DATA_BLOCK "HMI animation"	// DB 60
TITLE = HMI ANIMATION DATA BLOCK
AUTHOR : Milesi
VERSION : 0.1
  STRUCT
   Take_up_unit : STRUCT
    DB60_DBX0_0 : BOOL ;	//General alarm
    DB60_DBX0_1 : BOOL ;	//Driven pintle emergency
    DB60_DBX0_2 : BOOL ;	//Idle pintle emergency
    DB60_DBX0_3 : BOOL ;	//Bobbin down
    DB60_DBX0_4 : BOOL ;	//Speed reference right inversion
    DB60_DBX0_5 : BOOL ;	//Speed reference left inversion
    DB60_DBX0_6 : BOOL ;
    DB60_DBX0_7 : BOOL ;
    DB60_DBB1 : BYTE ;	//Motor status
    DB60_DBB2 : BYTE ;	//Motor blower status
    DB60_DBB3 : BYTE ;	//Traverse motor status
    DB60_DBB4 : BYTE ;	//Traverse motor blower status
    DB60_DBB5 : BYTE ;	//Bobbin driven pintle motor status
    DB60_DBB6 : BYTE ;	//Bobbin idle pintle motor status
    DB60_DBB7 : BYTE ;	//Bobbin pintle opening-closing motor status
    DB60_DBB8 : BYTE ;
    DB60_DBB9 : BYTE ;
    DB60_DBB10 : BYTE ;
   END_STRUCT ;
   Capstan : STRUCT
    DB60_DBX12_0 : BOOL ;	//General alarm
    DB60_DBX12_1 : BOOL ;	//Cable block open
    DB60_DBX12_2 : BOOL ;
    DB60_DBX12_3 : BOOL ;
    DB60_DBX12_4 : BOOL ;
    DB60_DBX12_5 : BOOL ;
    DB60_DBX12_6 : BOOL ;
    DB60_DBX12_7 : BOOL ;
    DB60_DBB13 : BYTE ;	//Motor status
    DB60_DBB14 : BYTE ;	//Motor blower status
    DB60_DBW16 : INT ;
    DB60_DBW18 : INT ;
    DB60_DBD20 : REAL ;
   END_STRUCT ;
   Lateral_taping_head : STRUCT
    DB60_DBX24_0 : BOOL ;	//General alarm
    DB60_DBX24_1 : BOOL ;
    DB60_DBX24_2 : BOOL ;
    DB60_DBX24_3 : BOOL ;
    DB60_DBX24_4 : BOOL ;
    DB60_DBX24_5 : BOOL ;
    DB60_DBX24_6 : BOOL ;
    DB60_DBX24_7 : BOOL ;
    DB60_DBB25 : BYTE ;	//Motor status
    DB60_DBB26 : BYTE ;	//Motor blower status
    DB60_DBW28 : INT ;
    DB60_DBW30 : INT ;
    DB60_DBD32 : REAL ;
   END_STRUCT ;
   Cage_24 : STRUCT
    DB60_DBX36_0 : BOOL ;	//General alarm
    DB60_DBX36_1 : BOOL ;
    DB60_DBX36_2 : BOOL ;
    DB60_DBX36_3 : BOOL ;
    DB60_DBX36_4 : BOOL ;
    DB60_DBX36_5 : BOOL ;
    DB60_DBX36_6 : BOOL ;
    DB60_DBX36_7 : BOOL ;
    DB60_DBB37 : BYTE ;	//Motor status
    DB60_DBB38 : BYTE ;	//Motor blower status
    DB60_DBB39 : BYTE ;	//Loading motor status
    DB60_DBB40 : BYTE ;
    DB60_DBW42 : INT ;
    DB60_DBD46 : REAL ;
   END_STRUCT ;
   Cage_24_preforming : STRUCT
    DB60_DBX48_0 : BOOL ;	//General alarm
    DB60_DBX48_1 : BOOL ;
    DB60_DBX48_2 : BOOL ;
    DB60_DBX48_3 : BOOL ;
    DB60_DBX48_4 : BOOL ;
    DB60_DBX48_5 : BOOL ;
    DB60_DBX48_6 : BOOL ;
    DB60_DBX48_7 : BOOL ;
    DB60_DBB49 : BYTE ;	//Motor status
    DB60_DBB50 : BYTE ;	//Motor blower status
    DB60_DBW52 : INT ;
    DB60_DBW54 : INT ;
    DB60_DBD56 : REAL ;
   END_STRUCT ;
   Cage_18 : STRUCT
    DB60_DBX60_0 : BOOL ;	//General alarm
    DB60_DBX60_1 : BOOL ;
    DB60_DBX60_2 : BOOL ;
    DB60_DBX60_3 : BOOL ;
    DB60_DBX60_4 : BOOL ;
    DB60_DBX60_5 : BOOL ;
    DB60_DBX60_6 : BOOL ;
    DB60_DBX60_7 : BOOL ;
    DB60_DBB61 : BYTE ;	//Motor status
    DB60_DBB62 : BYTE ;	//Motor blower status
    DB60_DBB63 : BYTE ;	//Loading motor status
    DB60_DBB64 : BYTE ;
    DB60_DBW66 : INT ;
    DB60_DBD68 : REAL ;
   END_STRUCT ;
   Cage_18_preforming : STRUCT
    DB60_DBX72_0 : BOOL ;	//General alarm
    DB60_DBX72_1 : BOOL ;
    DB60_DBX72_2 : BOOL ;
    DB60_DBX72_3 : BOOL ;
    DB60_DBX72_4 : BOOL ;
    DB60_DBX72_5 : BOOL ;
    DB60_DBX72_6 : BOOL ;
    DB60_DBX72_7 : BOOL ;
    DB60_DBB73 : BYTE ;	//Motor status
    DB60_DBB74 : BYTE ;	//Motor blower status
    DB60_DBW76 : INT ;
    DB60_DBW78 : INT ;
    DB60_DBD80 : REAL ;
   END_STRUCT ;
   Cage_12 : STRUCT
    DB60_DBX84_0 : BOOL ;	//General alarm
    DB60_DBX84_1 : BOOL ;
    DB60_DBX84_2 : BOOL ;
    DB60_DBX84_3 : BOOL ;
    DB60_DBX84_4 : BOOL ;
    DB60_DBX84_5 : BOOL ;
    DB60_DBX84_6 : BOOL ;
    DB60_DBX84_7 : BOOL ;
    DB60_DBB85 : BYTE ;	//Motor status
    DB60_DBB86 : BYTE ;	//Motor blower status
    DB60_DBB87 : BYTE ;	//Loading motor status
    DB60_DBB88 : BYTE ;
    DB60_DBW90 : INT ;
    DB60_DBD92 : REAL ;
   END_STRUCT ;
   Cage_12_preforming : STRUCT
    DB60_DBX96_0 : BOOL ;	//General alarm
    DB60_DBX96_1 : BOOL ;
    DB60_DBX96_2 : BOOL ;
    DB60_DBX96_3 : BOOL ;
    DB60_DBX96_4 : BOOL ;
    DB60_DBX96_5 : BOOL ;
    DB60_DBX96_6 : BOOL ;
    DB60_DBX96_7 : BOOL ;
    DB60_DBB97 : BYTE ;	//Motor status
    DB60_DBB98 : BYTE ;	//Motor blower status
    DB60_DBB99 : BYTE ;
    DB60_DBW100 : INT ;
    DB60_DBW102 : INT ;
    DB60_DBD104 : REAL ;
   END_STRUCT ;
   Cage_6 : STRUCT
    DB60_DBX108_0 : BOOL ;	//General alarm
    DB60_DBX108_1 : BOOL ;	//Preforming general alarm
    DB60_DBX108_2 : BOOL ;
    DB60_DBX108_3 : BOOL ;
    DB60_DBX108_4 : BOOL ;
    DB60_DBX108_5 : BOOL ;
    DB60_DBX108_6 : BOOL ;
    DB60_DBX108_7 : BOOL ;
    DB60_DBB109 : BYTE ;	//Motor status
    DB60_DBB110 : BYTE ;	//Motor blower status
    DB60_DBB111 : BYTE ;	//Loading motor status
    DB60_DBB112 : BYTE ;
    DB60_DBW114 : INT ;
    DB60_DBD116 : REAL ;
   END_STRUCT ;
   Cage_6_preforming : STRUCT
    DB60_DBX120_0 : BOOL ;	//General alarm
    DB60_DBX120_1 : BOOL ;
    DB60_DBX120_2 : BOOL ;
    DB60_DBX120_3 : BOOL ;
    DB60_DBX120_4 : BOOL ;
    DB60_DBX120_5 : BOOL ;
    DB60_DBX120_6 : BOOL ;
    DB60_DBX120_7 : BOOL ;
    DB60_DBB121 : BYTE ;
    DB60_DBB122 : BYTE ;
    DB60_DBW124 : INT ;
    DB60_DBW126 : INT ;
    DB60_DBD128 : REAL ;
   END_STRUCT ;
   Pay_off_630 : STRUCT
    DB60_DBX132_0 : BOOL ;	//General alarm
    DB60_DBX132_1 : BOOL ;	//Open pintles
    DB60_DBX132_2 : BOOL ;
    DB60_DBX132_3 : BOOL ;
    DB60_DBX132_4 : BOOL ;
    DB60_DBX132_5 : BOOL ;
    DB60_DBX132_6 : BOOL ;
    DB60_DBX132_7 : BOOL ;
    DB60_DBB133 : BYTE ;
    DB60_DBB134 : BYTE ;
    DB60_DBW136 : INT ;
    DB60_DBW138 : INT ;
    DB60_DBD140 : REAL ;
   END_STRUCT ;
   Pay_off_unit : STRUCT
    DB60_DBX144_0 : BOOL ;	//General alarm
    DB60_DBX144_1 : BOOL ;	//Driven pintle emergency
    DB60_DBX144_2 : BOOL ;	//Idle pintle emergency
    DB60_DBX144_3 : BOOL ;	//Bobbin down
    DB60_DBX144_4 : BOOL ;	//Right direction
    DB60_DBX144_5 : BOOL ;	//Left direction
    DB60_DBX144_6 : BOOL ;
    DB60_DBX144_7 : BOOL ;
    DB60_DBB145 : BYTE ;	//Traverse motor status
    DB60_DBB146 : BYTE ;	//Traverse motor blower status
    DB60_DBB147 : BYTE ;	//Bobbin driven pintle motor status
    DB60_DBB148 : BYTE ;	//Bobbin idle pintle motor status
    DB60_DBB149 : BYTE ;	//Bobbin pintle opening-closing motor status
    DB60_DBB150 : BYTE ;
    DB60_DBD152 : REAL ;
   END_STRUCT ;
   Line : STRUCT
    DB60_DBX156_0 : BOOL ;	//General alarm
    DB60_DBX156_1 : BOOL ;	//Alarms present to HMI
    DB60_DBX156_2 : BOOL ;	//Line run with zero speed to HMI
    DB60_DBX156_3 : BOOL ;
    DB60_DBX156_4 : BOOL ;
    DB60_DBX156_5 : BOOL ;
    DB60_DBX156_6 : BOOL ;
    DB60_DBX156_7 : BOOL ;	//PLC<--->HMI comunication on control
    DB60_DBB157 : BYTE ;
    DB60_DBB158 : BYTE ;
    DB60_DBW160 : INT ;
    DB60_DBW162 : INT ;
    DB60_DBD164 : REAL ;
   END_STRUCT ;
  END_STRUCT ;	
BEGIN
   Take_up_unit.DB60_DBX0_3 := TRUE;
   Take_up_unit.DB60_DBX0_5 := TRUE;
   Take_up_unit.DB60_DBB1 := B#16#1;
   Take_up_unit.DB60_DBB2 := B#16#1;
   Cage_24.DB60_DBX36_0 := TRUE;
   Cage_18.DB60_DBX60_0 := TRUE;
   Cage_6_preforming.DB60_DBX120_1 := TRUE;
   Cage_6_preforming.DB60_DBW126 := 465;
   Pay_off_630.DB60_DBX132_1 := TRUE;
   Pay_off_unit.DB60_DBX144_3 := TRUE;
   Pay_off_unit.DB60_DBB146 := B#16#1;
   Line.DB60_DBX156_7 := TRUE;
END_DATA_BLOCK

DATA_BLOCK "MAP_DI"	// DB 91
TITLE = Mappa Ingressi
VERSION : 0.0
  STRUCT
   DB91_DBX000_0 : BOOL ;	//Auxiliary on [-126K1|E000.0]
   DB91_DBX000_1 : BOOL ;	//Emergency push-buttons [-126K4|E000.1]
   DB91_DBX000_2 : BOOL ;	//Cabinet thermo-switch [-175S3|E000.2]
   DB91_DBX000_3 : BOOL ;	//Auxiliary 230v transformer overload [-112Q3|E000.3]
   DB91_DBX000_4 : BOOL ;	//24DC UPS module battery alarm [-108G1:Alarm|E000.4]
   DB91_DBX000_5 : BOOL ;	//24DC UPS module battery packs ok [-108G1:Bat ok|E000.5]
   DB91_DBX000_6 : BOOL ;	//Cabinet air fans overload [-116Q1|E000.6]
   DB91_DBX000_7 : BOOL ;
   DB91_DBX001_0 : BOOL ;	//Dryer supply overload [-119Q1|E001.0]
   DB91_DBX001_1 : BOOL ;	//Ac motor drives feeder braking resistor alarm [-141R1:T2|E001.1]
   DB91_DBX001_2 : BOOL ;	//Ac motor drives feeder dc bus alarm [-140G1:X104:20|E001.2]
   DB91_DBX001_3 : BOOL ;
   DB91_DBX001_4 : BOOL ;
   DB91_DBX001_5 : BOOL ;
   DB91_DBX001_6 : BOOL ;
   DB91_DBX001_7 : BOOL ;
   DB91_DBX002_0 : BOOL ;	//Line stop push-buttons [-177S1|E006.3]
   DB91_DBX002_1 : BOOL ;	//Line run push-buttons [-177S2|E006.4]
   DB91_DBX002_2 : BOOL ;	//Line jog push-buttons [-177S3|E006.5]
   DB91_DBX002_3 : BOOL ;	//Line alarms reset push-buttons [-177S4|E006.6]
   DB91_DBX002_4 : BOOL ;	//Hold line speed push-button [-177S5|E006.7]
   DB91_DBX002_5 : BOOL ;	//Power supply on [-112K1|E008.0]
   DB91_DBX002_6 : BOOL ;	//Power supply on end of time [-112K1:66|E008.1]
   DB91_DBX002_7 : BOOL ;	//230VAC UPS main failure [-113G1:4|E008.2]
   DB91_DBX003_0 : BOOL ;	//230VAC UPS battery nearly low [-113G1:3|E008.3]
   DB91_DBX003_1 : BOOL ;	//24DC aux. feeding overload [-109Q6|E008.4]
   DB91_DBX003_2 : BOOL ;	//preforming motor blower and inverter fan supply overload [-115Q1|E008.5]
   DB91_DBX003_3 : BOOL ;	//AC motor drive feeder fan overload [-140Q1|E008.6]
   DB91_DBX003_4 : BOOL ;	//24VDC PLC input supply overload [-109Q2|E008.7]
   DB91_DBX003_5 : BOOL ;
   DB91_DBX003_6 : BOOL ;
   DB91_DBX003_7 : BOOL ;
   DB91_DBX004_0 : BOOL ;	//Take-up bobbin increase pull push-button [-922S5|E001.7]
   DB91_DBX004_1 : BOOL ;	//Take-up bobbin decrease pull push-button [-922S6|E002.0]
   DB91_DBX004_2 : BOOL ;	//Take-up bobbin stop push-buttons [-922S7|E002.1]
   DB91_DBX004_3 : BOOL ;	//Take-up bobbin run push-buttons [-922S8|E002.2]
   DB91_DBX004_4 : BOOL ;	//Take-up bobbin motor blower overload [-945Q1|E037.3]
   DB91_DBX004_5 : BOOL ;	//Take-up bobbin motor electric brake overload [-941Q2|E037.0]
   DB91_DBX004_6 : BOOL ;	//Take-up bobbin forward jog selector-switch [-964S1:Forward|E036.0]
   DB91_DBX004_7 : BOOL ;	//Take-up bobbin backward jog selector-switch [-964S1:Backward|E036.1]
   DB91_DBX005_0 : BOOL ;
   DB91_DBX005_1 : BOOL ;
   DB91_DBX005_2 : BOOL ;
   DB91_DBX005_3 : BOOL ;
   DB91_DBX005_4 : BOOL ;
   DB91_DBX005_5 : BOOL ;
   DB91_DBX005_6 : BOOL ;
   DB91_DBX005_7 : BOOL ;
   DB91_DBX006_0 : BOOL ;	//Take-up idle pintle up limit-switch [-961S1|E032.0]
   DB91_DBX006_1 : BOOL ;	//Take-up idle pintle down limit-switch [-961S2|E032.1]
   DB91_DBX006_2 : BOOL ;	//Take-up driven pintle up limit-switch [-961S3|E032.2]
   DB91_DBX006_3 : BOOL ;	//Take-up driven pintle down limit-switch [-961S4|E032.3]
   DB91_DBX006_4 : BOOL ;	//Take-up driven pintle up selector-switch [-961S5:UP|E033.0]
   DB91_DBX006_5 : BOOL ;	//Take-up driven pintle down selector-switch [-961S5:DOWN|E033.1]
   DB91_DBX006_6 : BOOL ;	//Take-up idle pintle up selector-switch [-961S7:UP|E033.2]
   DB91_DBX006_7 : BOOL ;	//Take-up idle pintle down selector-switch [-961S7:DOWN|E033.3]
   DB91_DBX007_0 : BOOL ;	//Take-up pintles up selector-switches [-962S1:UP|E034.0]
   DB91_DBX007_1 : BOOL ;	//Take-up pintles down selector-switches [-962S1:DOWN|E034.1]
   DB91_DBX007_2 : BOOL ;	//Take-up idle pintle opening selector-switches [-962S3:OPEN|E034.2]
   DB91_DBX007_3 : BOOL ;	//Take-up idle pintle closing selector-switches [-962S3:CLOSE|E034.3]
   DB91_DBX007_4 : BOOL ;	//Take-up idle pintle emergency limit-switch [-962S5|E035.0]
   DB91_DBX007_5 : BOOL ;	//Take-up driven pintle emergency limit-switch [-962S6|E035.1]
   DB91_DBX007_6 : BOOL ;
   DB91_DBX007_7 : BOOL ;
   DB91_DBX008_0 : BOOL ;	//Take-up traverse quick left push-buttons local panel [-962S7|E035.2]
   DB91_DBX008_1 : BOOL ;	//Take-up traverse quick right push-buttons local panel [-962S8|E035.3]
   DB91_DBX008_2 : BOOL ;	//Take-up traverse quick left push-buttons main panel [-922S3|E001.3]
   DB91_DBX008_3 : BOOL ;	//Take-up traverse quick right push-buttons main panel [-922S4|E001.4]
   DB91_DBX008_4 : BOOL ;	//Take-up traverse translation zero point sensor [-964B3|E036.2]
   DB91_DBX008_5 : BOOL ;	//Take-up traverse inversion delay sensor [-964B4|E036.3]
   DB91_DBX008_6 : BOOL ;	//Take-up traverse motor blower overload [-945Q2|E037.1]
   DB91_DBX008_7 : BOOL ;
   DB91_DBX009_0 : BOOL ;
   DB91_DBX009_1 : BOOL ;	//Take-up ac motors overload [-944Q1|E037.2]
   DB91_DBX009_2 : BOOL ;	//Take-up 230vac power supply overload [-112Q8|E001.5]
   DB91_DBX009_3 : BOOL ;	//Take-up 24vdc power supply overload [-109Q7|E001.6]
   DB91_DBX009_4 : BOOL ;
   DB91_DBX009_5 : BOOL ;
   DB91_DBX009_6 : BOOL ;
   DB91_DBX009_7 : BOOL ;
   DB91_DBX010_0 : BOOL ;
   DB91_DBX010_1 : BOOL ;
   DB91_DBX010_2 : BOOL ;
   DB91_DBX010_3 : BOOL ;
   DB91_DBX010_4 : BOOL ;
   DB91_DBX010_5 : BOOL ;
   DB91_DBX010_6 : BOOL ;
   DB91_DBX010_7 : BOOL ;
   DB91_DBX011_0 : BOOL ;
   DB91_DBX011_1 : BOOL ;
   DB91_DBX011_2 : BOOL ;
   DB91_DBX011_3 : BOOL ;
   DB91_DBX011_4 : BOOL ;
   DB91_DBX011_5 : BOOL ;
   DB91_DBX011_6 : BOOL ;
   DB91_DBX011_7 : BOOL ;
   DB91_DBX012_0 : BOOL ;	//Capstan motor blower overload [-705Q1|E002.3]
   DB91_DBX012_1 : BOOL ;	//Capstan minimum air pressure pressure-switch [-718S4|E002.4]
   DB91_DBX012_2 : BOOL ;	//Capstan motor brake control pressure-switch [-718S5|E002.5]
   DB91_DBX012_3 : BOOL ;	//Capstan cable clock open sensor [-718B6|E002.6]
   DB91_DBX012_4 : BOOL ;	//Cable block opening selector-switch [-177S6|E002.7]
   DB91_DBX012_5 : BOOL ;	//Capstan forward jog selector-switch [-177S7:Forward|E003.0]
   DB91_DBX012_6 : BOOL ;	//Capstan backward jog selector-switch [-177S7:Backward|E003.1]
   DB91_DBX012_7 : BOOL ;
   DB91_DBX013_0 : BOOL ;
   DB91_DBX013_1 : BOOL ;
   DB91_DBX013_2 : BOOL ;
   DB91_DBX013_3 : BOOL ;
   DB91_DBX013_4 : BOOL ;
   DB91_DBX013_5 : BOOL ;
   DB91_DBX013_6 : BOOL ;
   DB91_DBX013_7 : BOOL ;
   DB91_DBX014_0 : BOOL ;
   DB91_DBX014_1 : BOOL ;
   DB91_DBX014_2 : BOOL ;
   DB91_DBX014_3 : BOOL ;
   DB91_DBX014_4 : BOOL ;
   DB91_DBX014_5 : BOOL ;
   DB91_DBX014_6 : BOOL ;
   DB91_DBX014_7 : BOOL ;
   DB91_DBX015_0 : BOOL ;
   DB91_DBX015_1 : BOOL ;
   DB91_DBX015_2 : BOOL ;
   DB91_DBX015_3 : BOOL ;
   DB91_DBX015_4 : BOOL ;
   DB91_DBX015_5 : BOOL ;
   DB91_DBX015_6 : BOOL ;
   DB91_DBX015_7 : BOOL ;
   DB91_DBX016_0 : BOOL ;
   DB91_DBX016_1 : BOOL ;
   DB91_DBX016_2 : BOOL ;
   DB91_DBX016_3 : BOOL ;
   DB91_DBX016_4 : BOOL ;
   DB91_DBX016_5 : BOOL ;
   DB91_DBX016_6 : BOOL ;
   DB91_DBX016_7 : BOOL ;
   DB91_DBX017_0 : BOOL ;
   DB91_DBX017_1 : BOOL ;
   DB91_DBX017_2 : BOOL ;
   DB91_DBX017_3 : BOOL ;
   DB91_DBX017_4 : BOOL ;
   DB91_DBX017_5 : BOOL ;
   DB91_DBX017_6 : BOOL ;
   DB91_DBX017_7 : BOOL ;
   DB91_DBX018_0 : BOOL ;	//Cage 24 230VAC supply overload [-640Q1|E007.0]
   DB91_DBX018_1 : BOOL ;	//Cage 24 24VDC supply overload [-109Q12|E007.1]
   DB91_DBX018_2 : BOOL ;	//Cage 24 loading motor overload [-605Q2|E007.2]
   DB91_DBX018_3 : BOOL ;	//Cage 24 motor blower overload [-605Q1|E007.3]
   DB91_DBX018_4 : BOOL ;	//Cage 24 preforming motor electric brake overload [-607Q2|E007.4]
   DB91_DBX018_5 : BOOL ;	//Cage 24 preforming motor blower overload [-607Q1|E007.5]
   DB91_DBX018_6 : BOOL ;
   DB91_DBX018_7 : BOOL ;	//Cage 24 guard  blower motor overload [-606Q1|E007.7]
   DB91_DBX019_0 : BOOL ;
   DB91_DBX019_1 : BOOL ;
   DB91_DBX019_2 : BOOL ;
   DB91_DBX019_3 : BOOL ;
   DB91_DBX019_4 : BOOL ;
   DB91_DBX019_5 : BOOL ;
   DB91_DBX019_6 : BOOL ;
   DB91_DBX019_7 : BOOL ;
   DB91_DBX020_0 : BOOL ;	//Cage 24 loading line presence of air pressure-switch [-661S1|E042.0]
   DB91_DBX020_1 : BOOL ;	//Cage 24 brake control pressure-switch [-661S2|E042.1]
   DB91_DBX020_2 : BOOL ;	//Cage 24 minimum air pressure pressure-switch [-661S3|E042.2]
   DB91_DBX020_3 : BOOL ;	//Cage 24 piston engaged into cage limit-switch [-661S4|E042.3]
   DB91_DBX020_4 : BOOL ;	//Cage 24 piston disingaged out of cage limit-switch [-661S5|E042.4]
   DB91_DBX020_5 : BOOL ;	//Cage 24 loading motor engaged sensor [-661S6|E042.5]
   DB91_DBX020_6 : BOOL ;	//Cage 24 loading motor disengaged sensor [-661S7|E042.6]
   DB91_DBX020_7 : BOOL ;	//Cage 24 air pipe  limit-switch [-661S8|E042.7]
   DB91_DBX021_0 : BOOL ;	//Cage 24 presence of bobbin photocell -loading- [-662B1|E043.0]
   DB91_DBX021_1 : BOOL ;	//Cage 24 loading stop photocell [-662B2|E043.1]
   DB91_DBX021_2 : BOOL ;	//Cage 24 break of wire from ring [-662S3|E043.2]
   DB91_DBX021_3 : BOOL ;	//Cage 24 front door limit-switch [-686Y1|E043.3]
   DB91_DBX021_4 : BOOL ;	//Cage 24 rear door limit-switches [-662S5|E043.4]
   DB91_DBX021_5 : BOOL ;	//Cage 24 front guard open limit-switch [-662S6|E043.5]
   DB91_DBX021_6 : BOOL ;	//Cage 24 front guard closed sensor [-662B7|E043.6]
   DB91_DBX021_7 : BOOL ;	//Cage 24 guard presence of man photocell [-662B8|E043.7]
   DB91_DBX022_0 : BOOL ;	//Cage 24 line stop push-button [-663S1|E044.0]
   DB91_DBX022_1 : BOOL ;	//Cage 24 line jog push-button [-663S2|E044.1]
   DB91_DBX022_2 : BOOL ;	//Cage 24 loading run push-button [-663S3|E044.2]
   DB91_DBX022_3 : BOOL ;	//Cage 24 alarms reset push-button [-663S4|E044.3]
   DB91_DBX022_4 : BOOL ;	//Cage 24 guard closing selector-switch [-663S5:CLOSING|E044.4]
   DB91_DBX022_5 : BOOL ;	//Cage 24 guard opening selector-switch [-663S5:OPENING|E044.5]
   DB91_DBX022_6 : BOOL ;	//Cage 24 pintles closing selector-switch [-663S7:CLOSING|E044.6]
   DB91_DBX022_7 : BOOL ;	//Cage 24 pintles opening selector-switch [-663S7:OPENING|E044.7]
   DB91_DBX023_0 : BOOL ;	//Cage 24 pintles locking system closing selector-switch [-664S1:CLOSING|E045.0]
   DB91_DBX023_1 : BOOL ;	//Cage 24 pintles locking system opening selector-switch [-664S1:OPENING|E045.1]
   DB91_DBX023_2 : BOOL ;
   DB91_DBX023_3 : BOOL ;
   DB91_DBX023_4 : BOOL ;
   DB91_DBX023_5 : BOOL ;
   DB91_DBX023_6 : BOOL ;	//Cage 24 loading insertion push-button [-664S7|E045.6]
   DB91_DBX023_7 : BOOL ;
   DB91_DBX024_0 : BOOL ;
   DB91_DBX024_1 : BOOL ;
   DB91_DBX024_2 : BOOL ;
   DB91_DBX024_3 : BOOL ;
   DB91_DBX024_4 : BOOL ;
   DB91_DBX024_5 : BOOL ;
   DB91_DBX024_6 : BOOL ;	//Cage 24 preforming guard limit-switch [-688Y8|E046.6]
   DB91_DBX024_7 : BOOL ;	//Cage 24 preforming brake release push-button [-665S8|E046.7]
   DB91_DBX025_0 : BOOL ;	//Cage 24 preforming line stop push-button [-666S1|E047.0]
   DB91_DBX025_1 : BOOL ;	//Cage 24 preforming line jog push-button [-666S2|E047.1]
   DB91_DBX025_2 : BOOL ;
   DB91_DBX025_3 : BOOL ;
   DB91_DBX025_4 : BOOL ;
   DB91_DBX025_5 : BOOL ;
   DB91_DBX025_6 : BOOL ;
   DB91_DBX025_7 : BOOL ;
   DB91_DBX026_0 : BOOL ;
   DB91_DBX026_1 : BOOL ;
   DB91_DBX026_2 : BOOL ;
   DB91_DBX026_3 : BOOL ;
   DB91_DBX026_4 : BOOL ;
   DB91_DBX026_5 : BOOL ;
   DB91_DBX026_6 : BOOL ;
   DB91_DBX026_7 : BOOL ;
   DB91_DBX027_0 : BOOL ;
   DB91_DBX027_1 : BOOL ;
   DB91_DBX027_2 : BOOL ;
   DB91_DBX027_3 : BOOL ;
   DB91_DBX027_4 : BOOL ;	//Cage 24 bobbin brakes air tank pressure switch [-670S1|E050.2]
   DB91_DBX027_5 : BOOL ;	//Cage 24 line 1 pintles open [-670S2|E050.3]
   DB91_DBX027_6 : BOOL ;	//Cage 24 line 2 pintles open [-670S3|E050.4]
   DB91_DBX027_7 : BOOL ;	//Cage 24 line 3 pintles open [-670S4|E050.5]
   DB91_DBX028_0 : BOOL ;
   DB91_DBX028_1 : BOOL ;
   DB91_DBX028_2 : BOOL ;
   DB91_DBX028_3 : BOOL ;
   DB91_DBX028_4 : BOOL ;
   DB91_DBX028_5 : BOOL ;
   DB91_DBX028_6 : BOOL ;
   DB91_DBX028_7 : BOOL ;
   DB91_DBX029_0 : BOOL ;
   DB91_DBX029_1 : BOOL ;
   DB91_DBX029_2 : BOOL ;
   DB91_DBX029_3 : BOOL ;
   DB91_DBX029_4 : BOOL ;
   DB91_DBX029_5 : BOOL ;
   DB91_DBX029_6 : BOOL ;
   DB91_DBX029_7 : BOOL ;
   DB91_DBX030_0 : BOOL ;	//Cage 24 bobbin 1 break of wire and diameter calculation [-667B1|E047.2]
   DB91_DBX030_1 : BOOL ;	//Cage 24 bobbin 2 break of wire [-667B2|E047.3]
   DB91_DBX030_2 : BOOL ;	//Cage 24 bobbin 3 break of wire [-667B3|E047.4]
   DB91_DBX030_3 : BOOL ;	//Cage 24 bobbin 4 break of wire [-667B4|E047.5]
   DB91_DBX030_4 : BOOL ;	//Cage 24 bobbin 5 break of wire [-667B5|E047.6]
   DB91_DBX030_5 : BOOL ;	//Cage 24 bobbin 6 break of wire [-667B6|E047.7]
   DB91_DBX030_6 : BOOL ;	//Cage 24 bobbin 7 break of wire [-667B7|E048.0]
   DB91_DBX030_7 : BOOL ;	//Cage 24 bobbin 8 break of wire [-667B8|E048.1]
   DB91_DBX031_0 : BOOL ;	//Cage 24 bobbin 9 break of wire [-668B1|E048.2]
   DB91_DBX031_1 : BOOL ;	//Cage 24 bobbin 10 break of wire [-668B2|E048.3]
   DB91_DBX031_2 : BOOL ;	//Cage 24 bobbin 11 break of wire [-668B3|E048.4]
   DB91_DBX031_3 : BOOL ;	//Cage 24 bobbin 12 break of wire [-668B4|E048.5]
   DB91_DBX031_4 : BOOL ;	//Cage 24 bobbin 13 break of wire [-668B5|E048.6]
   DB91_DBX031_5 : BOOL ;	//Cage 24 bobbin 14 break of wire [-668B6|E048.7]
   DB91_DBX031_6 : BOOL ;	//Cage 24 bobbin 15 break of wire [-668B7|E049.0]
   DB91_DBX031_7 : BOOL ;	//Cage 24 bobbin 16 break of wire [-668B8|E049.1]
   DB91_DBX032_0 : BOOL ;	//Cage 24 bobbin 17 break of wire [-669B1|E049.2]
   DB91_DBX032_1 : BOOL ;	//Cage 24 bobbin 18 break of wire [-669B2|E049.3]
   DB91_DBX032_2 : BOOL ;	//Cage 24 bobbin 19 break of wire [-669B3|E049.4]
   DB91_DBX032_3 : BOOL ;	//Cage 24 bobbin 20 break of wire [-669B4|E049.5]
   DB91_DBX032_4 : BOOL ;	//Cage 24 bobbin 21 break of wire [-669B5|E049.6]
   DB91_DBX032_5 : BOOL ;	//Cage 24 bobbin 22 break of wire [-669B6|E049.7]
   DB91_DBX032_6 : BOOL ;	//Cage 24 bobbin 23 break of wire [-669B7|E050.0]
   DB91_DBX032_7 : BOOL ;	//Cage 24 bobbin 24 break of wire [-669B8|E050.1]
   DB91_DBX033_0 : BOOL ;
   DB91_DBX033_1 : BOOL ;
   DB91_DBX033_2 : BOOL ;
   DB91_DBX033_3 : BOOL ;
   DB91_DBX033_4 : BOOL ;
   DB91_DBX033_5 : BOOL ;
   DB91_DBX033_6 : BOOL ;
   DB91_DBX033_7 : BOOL ;
   DB91_DBX034_0 : BOOL ;
   DB91_DBX034_1 : BOOL ;
   DB91_DBX034_2 : BOOL ;
   DB91_DBX034_3 : BOOL ;
   DB91_DBX034_4 : BOOL ;
   DB91_DBX034_5 : BOOL ;
   DB91_DBX034_6 : BOOL ;
   DB91_DBX034_7 : BOOL ;
   DB91_DBX035_0 : BOOL ;
   DB91_DBX035_1 : BOOL ;
   DB91_DBX035_2 : BOOL ;
   DB91_DBX035_3 : BOOL ;
   DB91_DBX035_4 : BOOL ;
   DB91_DBX035_5 : BOOL ;
   DB91_DBX035_6 : BOOL ;
   DB91_DBX035_7 : BOOL ;
   DB91_DBX036_0 : BOOL ;	//Cage 24 Loader in stand by zone [+MCB24:7|E010.4]
   DB91_DBX036_1 : BOOL ;	//Cage 24 Loader inside cage [+MCB24:8|E010.5]
   DB91_DBX036_2 : BOOL ;	//Cage 24 Loader open clamp [+MCB24:9|E010.6]
   DB91_DBX036_3 : BOOL ;	//Cage 24 Loader to parcking zone [+MCB24:10|E010.7]
   DB91_DBX036_4 : BOOL ;
   DB91_DBX036_5 : BOOL ;
   DB91_DBX036_6 : BOOL ;
   DB91_DBX036_7 : BOOL ;
   DB91_DBX037_0 : BOOL ;
   DB91_DBX037_1 : BOOL ;
   DB91_DBX037_2 : BOOL ;
   DB91_DBX037_3 : BOOL ;
   DB91_DBX037_4 : BOOL ;
   DB91_DBX037_5 : BOOL ;
   DB91_DBX037_6 : BOOL ;
   DB91_DBX037_7 : BOOL ;
   DB91_DBX038_0 : BOOL ;	//Cage 18 230vac power supply overload [-540Q1|E003.2]
   DB91_DBX038_1 : BOOL ;	//Cage 18 24vdc power supply overload [-109Q11|E003.3]
   DB91_DBX038_2 : BOOL ;	//Cage 18 loading motor overload [-505Q2|E003.4]
   DB91_DBX038_3 : BOOL ;	//Cage 18 motor blower overload [-505Q1|E003.5]
   DB91_DBX038_4 : BOOL ;	//Cage 18 preforming motor electric brake overload [-507Q2|E003.6]
   DB91_DBX038_5 : BOOL ;	//Cage 18 preforming motor blower overload [-507Q1|E003.7]
   DB91_DBX038_6 : BOOL ;
   DB91_DBX038_7 : BOOL ;	//Cage 18 guard blower motor overload [-506Q1|E004.1]
   DB91_DBX039_0 : BOOL ;
   DB91_DBX039_1 : BOOL ;
   DB91_DBX039_2 : BOOL ;
   DB91_DBX039_3 : BOOL ;
   DB91_DBX039_4 : BOOL ;
   DB91_DBX039_5 : BOOL ;
   DB91_DBX039_6 : BOOL ;
   DB91_DBX039_7 : BOOL ;
   DB91_DBX040_0 : BOOL ;	//Cage 18 loading line presence of air pressure-switch [-561S1|E052.0]
   DB91_DBX040_1 : BOOL ;	//Cage 18 brake control pressure-switch [-561S2|E052.1]
   DB91_DBX040_2 : BOOL ;	//Cage 18 minimum air pressure pressure-switch [-561S3|E052.2]
   DB91_DBX040_3 : BOOL ;	//Cage 18 piston engaged in cage limit-switch [-561S4|E052.3]
   DB91_DBX040_4 : BOOL ;	//Cage 18 piston disengaged from cage limit-switch [-561S5|E052.4]
   DB91_DBX040_5 : BOOL ;	//Cage 18 loading motor engaged sensor [-561B6|E052.5]
   DB91_DBX040_6 : BOOL ;	//Cage 18 loading motor disengaged sensor [-561B7|E052.6]
   DB91_DBX040_7 : BOOL ;	//Cage 18 air pipe limit-switch [-561S8|E052.7]
   DB91_DBX041_0 : BOOL ;	//Cage 18 presence of bobbin photocell -loading- [-562B1|E053.0]
   DB91_DBX041_1 : BOOL ;	//Cage 18 loading stop photocell [-562B2|E053.1]
   DB91_DBX041_2 : BOOL ;	//Cage 18 break of wire from ring [-562S3|E053.2]
   DB91_DBX041_3 : BOOL ;	//Cage 18 front door limit-switch [-586Y1|E053.3]
   DB91_DBX041_4 : BOOL ;	//Cage 18 rear doors limit-switches [-562S5|E053.4]
   DB91_DBX041_5 : BOOL ;	//Cage 18 front guard open limit-switch [-562S6|E053.5]
   DB91_DBX041_6 : BOOL ;	//Cage 18 front guard closed sensor [-562B7|E053.6]
   DB91_DBX041_7 : BOOL ;	//Cage 18 guard presence of man photocell [-562B8|E053.7]
   DB91_DBX042_0 : BOOL ;	//Cage 18 line stop push-button [-563S1|E054.0]
   DB91_DBX042_1 : BOOL ;	//Cage 18 line jog push-button [-563S2|E054.1]
   DB91_DBX042_2 : BOOL ;	//Cage 18 loading run push-button [-563S3|E054.2]
   DB91_DBX042_3 : BOOL ;	//Cage 18 alarms reset push-button [-563S4|E054.3]
   DB91_DBX042_4 : BOOL ;	//Cage 18 guard closing selector-switch [-563S5:CLOSING|E054.4]
   DB91_DBX042_5 : BOOL ;	//Cage 18 guard opening selector-switch [-563S5:OPENING|E054.5]
   DB91_DBX042_6 : BOOL ;	//Cage 18 pintles closing selector-switch [-563S7:CLOSING|E054.6]
   DB91_DBX042_7 : BOOL ;	//Cage 18 pintles opening selector-switch [-563S7:OPENING|E054.7]
   DB91_DBX043_0 : BOOL ;	//Cage 18 pintles locking system closing selector-switch [-564S1:CLOSING|E055.0]
   DB91_DBX043_1 : BOOL ;	//Cage 18 pintles locking system opening selector-switch [-563S1:OPENING|E055.1]
   DB91_DBX043_2 : BOOL ;
   DB91_DBX043_3 : BOOL ;
   DB91_DBX043_4 : BOOL ;
   DB91_DBX043_5 : BOOL ;
   DB91_DBX043_6 : BOOL ;	//Cage 18 loading insertion push-button [-564S7|E055.6]
   DB91_DBX043_7 : BOOL ;
   DB91_DBX044_0 : BOOL ;
   DB91_DBX044_1 : BOOL ;
   DB91_DBX044_2 : BOOL ;
   DB91_DBX044_3 : BOOL ;
   DB91_DBX044_4 : BOOL ;
   DB91_DBX044_5 : BOOL ;
   DB91_DBX044_6 : BOOL ;	//Cage 18 preforming guard limit-switch [-588Y8|E056.6]
   DB91_DBX044_7 : BOOL ;	//Cage 18 preforming brake release push-button [-565S8|E056.7]
   DB91_DBX045_0 : BOOL ;	//Cage 18 preforming line stop push-button [-566S1|E057.0]
   DB91_DBX045_1 : BOOL ;	//Cage 18 preforming line jog push-button [-566S2|E057.1]
   DB91_DBX045_2 : BOOL ;
   DB91_DBX045_3 : BOOL ;
   DB91_DBX045_4 : BOOL ;
   DB91_DBX045_5 : BOOL ;
   DB91_DBX045_6 : BOOL ;
   DB91_DBX045_7 : BOOL ;
   DB91_DBX046_0 : BOOL ;
   DB91_DBX046_1 : BOOL ;
   DB91_DBX046_2 : BOOL ;
   DB91_DBX046_3 : BOOL ;
   DB91_DBX046_4 : BOOL ;
   DB91_DBX046_5 : BOOL ;
   DB91_DBX046_6 : BOOL ;
   DB91_DBX046_7 : BOOL ;
   DB91_DBX047_0 : BOOL ;	//Cage 18 bobbin brakes air tank minimum pressure pressure-switch [-569S3|E059.4]
   DB91_DBX047_1 : BOOL ;	//Cage 18 line 1 pintles open [-569S4|E059.5]
   DB91_DBX047_2 : BOOL ;	//Cage 18 line 2 pintles open [-569S5|E059.6]
   DB91_DBX047_3 : BOOL ;	//Cage 18 line 3 pintles open [-569S6|E059.7]
   DB91_DBX047_4 : BOOL ;
   DB91_DBX047_5 : BOOL ;
   DB91_DBX047_6 : BOOL ;
   DB91_DBX047_7 : BOOL ;
   DB91_DBX048_0 : BOOL ;
   DB91_DBX048_1 : BOOL ;
   DB91_DBX048_2 : BOOL ;
   DB91_DBX048_3 : BOOL ;
   DB91_DBX048_4 : BOOL ;
   DB91_DBX048_5 : BOOL ;
   DB91_DBX048_6 : BOOL ;
   DB91_DBX048_7 : BOOL ;
   DB91_DBX049_0 : BOOL ;
   DB91_DBX049_1 : BOOL ;
   DB91_DBX049_2 : BOOL ;
   DB91_DBX049_3 : BOOL ;
   DB91_DBX049_4 : BOOL ;
   DB91_DBX049_5 : BOOL ;
   DB91_DBX049_6 : BOOL ;
   DB91_DBX049_7 : BOOL ;
   DB91_DBX050_0 : BOOL ;	//Cage 18 bobbin 1 break of wire and diameter calculation [-567B1|E057.2]
   DB91_DBX050_1 : BOOL ;	//Cage 18 bobbin 2 break of wire [-567B2|E057.3]
   DB91_DBX050_2 : BOOL ;	//Cage 18 bobbin 3 break of wire [-567B3|E057.4]
   DB91_DBX050_3 : BOOL ;	//Cage 18 bobbin 4 break of wire [-567B4|E057.5]
   DB91_DBX050_4 : BOOL ;	//Cage 18 bobbin 5 break of wire [-567B5|E057.6]
   DB91_DBX050_5 : BOOL ;	//Cage 18 bobbin 6 break of wire [-567B6|E057.7]
   DB91_DBX050_6 : BOOL ;	//Cage 18 bobbin 7 break of wire [-567B7|E058.0]
   DB91_DBX050_7 : BOOL ;	//Cage 18 bobbin 8 break of wire [-567B8|E058.1]
   DB91_DBX051_0 : BOOL ;	//Cage 18 bobbin 9 break of wire [-568B1|E058.2]
   DB91_DBX051_1 : BOOL ;	//Cage 18 bobbin 10 break of wire [-568B2|E058.3]
   DB91_DBX051_2 : BOOL ;	//Cage 18 bobbin 11 break of wire [-568B3|E058.4]
   DB91_DBX051_3 : BOOL ;	//Cage 18 bobbin 12 break of wire [-568B4|E058.5]
   DB91_DBX051_4 : BOOL ;	//Cage 18 bobbin 13 break of wire [-568B5|E058.6]
   DB91_DBX051_5 : BOOL ;	//Cage 18 bobbin 14 break of wire [-568B6|E058.7]
   DB91_DBX051_6 : BOOL ;	//Cage 18 bobbin 15 break of wire [-568B7|E059.0]
   DB91_DBX051_7 : BOOL ;	//Cage 18 bobbin 16 break of wire [-568B8|E059.1]
   DB91_DBX052_0 : BOOL ;	//Cage 18 bobbin 17 break of wire [-569B1|E059.2]
   DB91_DBX052_1 : BOOL ;	//Cage 18 bobbin 18 break of wire [-569B2|E059.3]
   DB91_DBX052_2 : BOOL ;
   DB91_DBX052_3 : BOOL ;
   DB91_DBX052_4 : BOOL ;
   DB91_DBX052_5 : BOOL ;
   DB91_DBX052_6 : BOOL ;
   DB91_DBX052_7 : BOOL ;
   DB91_DBX053_0 : BOOL ;
   DB91_DBX053_1 : BOOL ;
   DB91_DBX053_2 : BOOL ;
   DB91_DBX053_3 : BOOL ;
   DB91_DBX053_4 : BOOL ;
   DB91_DBX053_5 : BOOL ;
   DB91_DBX053_6 : BOOL ;
   DB91_DBX053_7 : BOOL ;
   DB91_DBX054_0 : BOOL ;
   DB91_DBX054_1 : BOOL ;
   DB91_DBX054_2 : BOOL ;
   DB91_DBX054_3 : BOOL ;
   DB91_DBX054_4 : BOOL ;
   DB91_DBX054_5 : BOOL ;
   DB91_DBX054_6 : BOOL ;
   DB91_DBX054_7 : BOOL ;
   DB91_DBX055_0 : BOOL ;
   DB91_DBX055_1 : BOOL ;
   DB91_DBX055_2 : BOOL ;
   DB91_DBX055_3 : BOOL ;
   DB91_DBX055_4 : BOOL ;
   DB91_DBX055_5 : BOOL ;
   DB91_DBX055_6 : BOOL ;
   DB91_DBX055_7 : BOOL ;
   DB91_DBX056_0 : BOOL ;	//Cage 18 Loader in stand by zone [+MCB18:7|E010.0]
   DB91_DBX056_1 : BOOL ;	//Cage 18 Loader inside cage [+MCB18:8|E010.1]
   DB91_DBX056_2 : BOOL ;	//Cage 18 Loader open clamp [+MCB18:9|E010.2]
   DB91_DBX056_3 : BOOL ;	//Cage 18 Loader to parcking zone [+MCB18:10|E010.3]
   DB91_DBX056_4 : BOOL ;	//Cage 18 Loader Locked [-565B5|E056.4]
   DB91_DBX056_5 : BOOL ;	//Cage 18 Loader UnLocked [-565B6|E056.5]
   DB91_DBX056_6 : BOOL ;
   DB91_DBX056_7 : BOOL ;
   DB91_DBX057_0 : BOOL ;	//Cage 18 loader locked
   DB91_DBX057_1 : BOOL ;	//Cage 18 loader unlocked
   DB91_DBX057_2 : BOOL ;
   DB91_DBX057_3 : BOOL ;
   DB91_DBX057_4 : BOOL ;
   DB91_DBX057_5 : BOOL ;
   DB91_DBX057_6 : BOOL ;
   DB91_DBX057_7 : BOOL ;
   DB91_DBX058_0 : BOOL ;	//Cage 12 230vac power supply overload [-440Q1|E004.2]
   DB91_DBX058_1 : BOOL ;	//Cage 12 24vdc power supply overload [-109Q10|E004.3]
   DB91_DBX058_2 : BOOL ;	//Cage 12 loading motor overload [-405Q2|E004.4]
   DB91_DBX058_3 : BOOL ;	//Cage 12 motor blower overload [-405Q1|E004.5]
   DB91_DBX058_4 : BOOL ;	//Cage 12 preforming motor electric brake overload [-407Q2|E004.6]
   DB91_DBX058_5 : BOOL ;	//Cage 12 preforming motor blower overload [-407Q1|E004.7]
   DB91_DBX058_6 : BOOL ;
   DB91_DBX058_7 : BOOL ;	//Cage 12 guard blower motor overload [-406Q1|E005.1]
   DB91_DBX059_0 : BOOL ;
   DB91_DBX059_1 : BOOL ;
   DB91_DBX059_2 : BOOL ;
   DB91_DBX059_3 : BOOL ;
   DB91_DBX059_4 : BOOL ;
   DB91_DBX059_5 : BOOL ;
   DB91_DBX059_6 : BOOL ;
   DB91_DBX059_7 : BOOL ;
   DB91_DBX060_0 : BOOL ;	//Cage 12 loading line presence of air pressure-switch [-461S1|E062.0]
   DB91_DBX060_1 : BOOL ;	//Cage 12 brake control pressure-switch [-461S2|E062.1]
   DB91_DBX060_2 : BOOL ;	//Cage 12 minimum air pressure pressure-switch [-461S3|E062.2]
   DB91_DBX060_3 : BOOL ;	//Cage 12 piston engaged in cage limit-switch [-461S4|E062.3]
   DB91_DBX060_4 : BOOL ;	//Cage 12 piston disengaged from cage limit-switch [-461S5|E062.4]
   DB91_DBX060_5 : BOOL ;	//Cage 12 loading motor engaged sensor [-461B6|E062.5]
   DB91_DBX060_6 : BOOL ;	//Cage 12 loading motor disengaged sensor [-461B7|E062.6]
   DB91_DBX060_7 : BOOL ;	//Cage 12 air pipe limit-switch [-461S8|E062.7]
   DB91_DBX061_0 : BOOL ;	//Cage 12 presence of bobbin photocell -loading- [-462B1|E063.0]
   DB91_DBX061_1 : BOOL ;	//Cage 12 loading stop photocell [-462B2|E063.1]
   DB91_DBX061_2 : BOOL ;	//Cage 12 break of wire from ring [-462S3|E063.2]
   DB91_DBX061_3 : BOOL ;	//Cage 12 front door limit-switch [-486Y1|E063.3]
   DB91_DBX061_4 : BOOL ;	//Cage 12 rear doors limit-switches [-462S5|E063.4]
   DB91_DBX061_5 : BOOL ;	//Cage 12 front guard open limit-switch [-462S6|E063.5]
   DB91_DBX061_6 : BOOL ;	//Cage 12 front guard closed sensor [-462B7|E063.6]
   DB91_DBX061_7 : BOOL ;	//Cage 12 guard presence of man photocell [-462B8|E063.7]
   DB91_DBX062_0 : BOOL ;	//Cage 12 line stop push-button [-463S1|E064.0]
   DB91_DBX062_1 : BOOL ;	//Cage 12 line jog push-button [-463S2|E064.1]
   DB91_DBX062_2 : BOOL ;	//Cage 12 loading run push-button [-463S3|E064.2]
   DB91_DBX062_3 : BOOL ;	//Cage 12 alarms reset push-button [-463S4|E064.3]
   DB91_DBX062_4 : BOOL ;	//Cage 12 guard closing selector-switch [-463S5:CLOSING|E064.4]
   DB91_DBX062_5 : BOOL ;	//Cage 12 guard opening selector-switch [-463S5:OPENING|E064.5]
   DB91_DBX062_6 : BOOL ;	//Cage 12 pintles closing selector-switch [-463S7:CLOSING|E064.6]
   DB91_DBX062_7 : BOOL ;	//Cage 12 pintles opening selector-switch [-463S7:OPENING|E064.7]
   DB91_DBX063_0 : BOOL ;	//Cage 12 pintles locking system closing selector-switch [-464S1:CLOSING|E065.0]
   DB91_DBX063_1 : BOOL ;	//Cage 12 pintles locking system opening selector-switch [-464S1:OPENING|E065.1]
   DB91_DBX063_2 : BOOL ;
   DB91_DBX063_3 : BOOL ;
   DB91_DBX063_4 : BOOL ;
   DB91_DBX063_5 : BOOL ;
   DB91_DBX063_6 : BOOL ;	//Cage 12 loading insertion push-button [-464S7|E065.6]
   DB91_DBX063_7 : BOOL ;
   DB91_DBX064_0 : BOOL ;
   DB91_DBX064_1 : BOOL ;
   DB91_DBX064_2 : BOOL ;
   DB91_DBX064_3 : BOOL ;
   DB91_DBX064_4 : BOOL ;
   DB91_DBX064_5 : BOOL ;
   DB91_DBX064_6 : BOOL ;	//Cage 12 preforming guard limit-switch [-488Y8|E066.6]
   DB91_DBX064_7 : BOOL ;	//Cage 12 preforming brake release push-button [-465S8|E066.7]
   DB91_DBX065_0 : BOOL ;	//Cage 12 preforming line stop push-button [-466S1|E067.0]
   DB91_DBX065_1 : BOOL ;	//Cage 12 preforming line jog push-button [-466S2|E067.1]
   DB91_DBX065_2 : BOOL ;
   DB91_DBX065_3 : BOOL ;
   DB91_DBX065_4 : BOOL ;
   DB91_DBX065_5 : BOOL ;
   DB91_DBX065_6 : BOOL ;
   DB91_DBX065_7 : BOOL ;
   DB91_DBX066_0 : BOOL ;
   DB91_DBX066_1 : BOOL ;
   DB91_DBX066_2 : BOOL ;
   DB91_DBX066_3 : BOOL ;
   DB91_DBX066_4 : BOOL ;
   DB91_DBX066_5 : BOOL ;
   DB91_DBX066_6 : BOOL ;
   DB91_DBX066_7 : BOOL ;
   DB91_DBX067_0 : BOOL ;	//Cage 12 bobbin brakes air tank minimum pressure pressure-switch [-468S5|E068.6]
   DB91_DBX067_1 : BOOL ;	//Cage 12 line 1 pintles open [-468S6|E068.7]
   DB91_DBX067_2 : BOOL ;	//Cage 12 line 2 pintles open [-468S7|E069.0]
   DB91_DBX067_3 : BOOL ;	//Cage 12 line 3 pintles open [-468S8|E069.1]
   DB91_DBX067_4 : BOOL ;
   DB91_DBX067_5 : BOOL ;
   DB91_DBX067_6 : BOOL ;
   DB91_DBX067_7 : BOOL ;
   DB91_DBX068_0 : BOOL ;
   DB91_DBX068_1 : BOOL ;
   DB91_DBX068_2 : BOOL ;
   DB91_DBX068_3 : BOOL ;
   DB91_DBX068_4 : BOOL ;
   DB91_DBX068_5 : BOOL ;
   DB91_DBX068_6 : BOOL ;
   DB91_DBX068_7 : BOOL ;
   DB91_DBX069_0 : BOOL ;
   DB91_DBX069_1 : BOOL ;
   DB91_DBX069_2 : BOOL ;
   DB91_DBX069_3 : BOOL ;
   DB91_DBX069_4 : BOOL ;
   DB91_DBX069_5 : BOOL ;
   DB91_DBX069_6 : BOOL ;
   DB91_DBX069_7 : BOOL ;
   DB91_DBX070_0 : BOOL ;	//Cage 12 bobbin 1 break of wire and diameter calculation [-467B1|E067.2]
   DB91_DBX070_1 : BOOL ;	//Cage 12 bobbin 2 break of wire [-467B2|E067.3]
   DB91_DBX070_2 : BOOL ;	//Cage 12 bobbin 3 break of wire [-467B3|E067.4]
   DB91_DBX070_3 : BOOL ;	//Cage 12 bobbin 4 break of wire [-467B4|E067.5]
   DB91_DBX070_4 : BOOL ;	//Cage 12 bobbin 5 break of wire [-467B5|E067.6]
   DB91_DBX070_5 : BOOL ;	//Cage 12 bobbin 6 break of wire [-467B6|E067.7]
   DB91_DBX070_6 : BOOL ;	//Cage 12 bobbin 7 break of wire [-467B7|E068.0]
   DB91_DBX070_7 : BOOL ;	//Cage 12 bobbin 8 break of wire [-467B8|E068.1]
   DB91_DBX071_0 : BOOL ;	//Cage 12 bobbin 9 break of wire [-468B1|E068.2]
   DB91_DBX071_1 : BOOL ;	//Cage 12 bobbin 10 break of wire [-468B2|E068.3]
   DB91_DBX071_2 : BOOL ;	//Cage 12 bobbin 11 break of wire [-468B3|E068.4]
   DB91_DBX071_3 : BOOL ;	//Cage 12 bobbin 12 break of wire [-468B4|E068.5]
   DB91_DBX071_4 : BOOL ;
   DB91_DBX071_5 : BOOL ;
   DB91_DBX071_6 : BOOL ;
   DB91_DBX071_7 : BOOL ;
   DB91_DBX072_0 : BOOL ;
   DB91_DBX072_1 : BOOL ;
   DB91_DBX072_2 : BOOL ;
   DB91_DBX072_3 : BOOL ;
   DB91_DBX072_4 : BOOL ;
   DB91_DBX072_5 : BOOL ;
   DB91_DBX072_6 : BOOL ;
   DB91_DBX072_7 : BOOL ;
   DB91_DBX073_0 : BOOL ;
   DB91_DBX073_1 : BOOL ;
   DB91_DBX073_2 : BOOL ;
   DB91_DBX073_3 : BOOL ;
   DB91_DBX073_4 : BOOL ;
   DB91_DBX073_5 : BOOL ;
   DB91_DBX073_6 : BOOL ;
   DB91_DBX073_7 : BOOL ;
   DB91_DBX074_0 : BOOL ;
   DB91_DBX074_1 : BOOL ;
   DB91_DBX074_2 : BOOL ;
   DB91_DBX074_3 : BOOL ;
   DB91_DBX074_4 : BOOL ;
   DB91_DBX074_5 : BOOL ;
   DB91_DBX074_6 : BOOL ;
   DB91_DBX074_7 : BOOL ;
   DB91_DBX075_0 : BOOL ;
   DB91_DBX075_1 : BOOL ;
   DB91_DBX075_2 : BOOL ;
   DB91_DBX075_3 : BOOL ;
   DB91_DBX075_4 : BOOL ;
   DB91_DBX075_5 : BOOL ;
   DB91_DBX075_6 : BOOL ;
   DB91_DBX075_7 : BOOL ;
   DB91_DBX076_0 : BOOL ;	//Cage 12 Loader in stand by zone [+MCB12:7|E009.4]
   DB91_DBX076_1 : BOOL ;	//Cage 12 Loader inside cage [+MCB12:8|E009.5]
   DB91_DBX076_2 : BOOL ;	//Cage 12 Loader open clamp [+MCB12:9|E009.6]
   DB91_DBX076_3 : BOOL ;	//Cage 12 Loader to parcking zone [+MCB12:10|E009.7]
   DB91_DBX076_4 : BOOL ;
   DB91_DBX076_5 : BOOL ;
   DB91_DBX076_6 : BOOL ;
   DB91_DBX076_7 : BOOL ;
   DB91_DBX077_0 : BOOL ;	//Cage 12 loader locked
   DB91_DBX077_1 : BOOL ;	//Cage 12 loader unlocked
   DB91_DBX077_2 : BOOL ;
   DB91_DBX077_3 : BOOL ;
   DB91_DBX077_4 : BOOL ;
   DB91_DBX077_5 : BOOL ;
   DB91_DBX077_6 : BOOL ;
   DB91_DBX077_7 : BOOL ;
   DB91_DBX078_0 : BOOL ;
   DB91_DBX078_1 : BOOL ;
   DB91_DBX078_2 : BOOL ;	//Cage 6 230vac power supply overload [-340Q1|E005.2]
   DB91_DBX078_3 : BOOL ;	//Cage 6 24vdc power supply overload [-109Q9|E005.3]
   DB91_DBX078_4 : BOOL ;	//Cage 6 loading motor overload [-305Q2|E005.4]
   DB91_DBX078_5 : BOOL ;	//Cage 6 motor blower overload [-305Q1|E005.5]
   DB91_DBX078_6 : BOOL ;
   DB91_DBX078_7 : BOOL ;	//Cage 6 guard blower motor overload [-306Q1|E005.7]
   DB91_DBX079_0 : BOOL ;
   DB91_DBX079_1 : BOOL ;
   DB91_DBX079_2 : BOOL ;
   DB91_DBX079_3 : BOOL ;
   DB91_DBX079_4 : BOOL ;
   DB91_DBX079_5 : BOOL ;
   DB91_DBX079_6 : BOOL ;
   DB91_DBX079_7 : BOOL ;
   DB91_DBX080_0 : BOOL ;	//Cage 6 loading line presence of air pressure-switch [-361S1|E072.0]
   DB91_DBX080_1 : BOOL ;	//Cage 6 brake control pressure-switch [-361S2|E072.1]
   DB91_DBX080_2 : BOOL ;	//Cage 6 minimum air pressure pressure-switch [-361S3|E072.2]
   DB91_DBX080_3 : BOOL ;	//Cage 6 piston engaged in cage limit-switch [-361S4|E072.3]
   DB91_DBX080_4 : BOOL ;	//Cage 6 piston disengaged from cage limit-switch [-361S5|E072.4]
   DB91_DBX080_5 : BOOL ;	//Cage 6 loading motor engaged sensor [-361B6|E072.5]
   DB91_DBX080_6 : BOOL ;	//Cage 6 loading motor disengaged sensor [-361B7|E072.6]
   DB91_DBX080_7 : BOOL ;	//Cage 6 air pipe limit-switch [-361S8|E072.7]
   DB91_DBX081_0 : BOOL ;	//Cage 6 presence of bobbin photocell -loading- [-361B1|E073.0]
   DB91_DBX081_1 : BOOL ;	//Cage 6 loading stop photocell [-362B2|E073.1]
   DB91_DBX081_2 : BOOL ;	//Cage 6 break of wire from ring [-362S3|E073.2]
   DB91_DBX081_3 : BOOL ;	//Cage 6 front door limit-switch [-386Y1|E073.3]
   DB91_DBX081_4 : BOOL ;	//Cage 6 rear doors limit-switches [-362S5|E073.4]
   DB91_DBX081_5 : BOOL ;	//Cage 6 front guard open limit-switch [-362S6|E073.5]
   DB91_DBX081_6 : BOOL ;	//Cage 6 front guard closed sensor [-362B7|E073.6]
   DB91_DBX081_7 : BOOL ;	//Cage 6 guard presence of man photocell [-362B8|E073.7]
   DB91_DBX082_0 : BOOL ;	//Cage 6 line stop push-button [-363S1|E074.0]
   DB91_DBX082_1 : BOOL ;	//Cage 6 line jog push-button [-363S2|E074.1]
   DB91_DBX082_2 : BOOL ;	//Cage 6 loading run push-button [-363S3|E074.2]
   DB91_DBX082_3 : BOOL ;	//Cage 6 alarms reset push-button [-363S4|E074.3]
   DB91_DBX082_4 : BOOL ;	//Cage 6 guard closing selector-switch [-363S5:CLOSING|E074.4]
   DB91_DBX082_5 : BOOL ;	//Cage 6 guard opening selector-switch [-363S5:OPENING|E074.5]
   DB91_DBX082_6 : BOOL ;	//Cage 6 pintles closing selector-switch [-363S7:CLOSING|E074.6]
   DB91_DBX082_7 : BOOL ;	//Cage 6 pintles opening selector-switch [-363S7:OPENING|E074.7]
   DB91_DBX083_0 : BOOL ;	//Cage 6 pintles locking system closing selector-switch [-364S1:Closing|E075.0]
   DB91_DBX083_1 : BOOL ;	//Cage 6 pintles locking system opening selector-switch [-364S1:Opening|E075.1]
   DB91_DBX083_2 : BOOL ;
   DB91_DBX083_3 : BOOL ;
   DB91_DBX083_4 : BOOL ;
   DB91_DBX083_5 : BOOL ;
   DB91_DBX083_6 : BOOL ;	//Cage 6 loading insertion push-button [-364S7|E075.6]
   DB91_DBX083_7 : BOOL ;
   DB91_DBX084_0 : BOOL ;
   DB91_DBX084_1 : BOOL ;
   DB91_DBX084_2 : BOOL ;
   DB91_DBX084_3 : BOOL ;
   DB91_DBX084_4 : BOOL ;
   DB91_DBX084_5 : BOOL ;
   DB91_DBX084_6 : BOOL ;	//Cage 6 preforming guard limit-switch [-388Y8|E076.6]
   DB91_DBX084_7 : BOOL ;
   DB91_DBX085_0 : BOOL ;	//Cage 6 preforming line stop push-button [-365S|E076.7]
   DB91_DBX085_1 : BOOL ;	//Cage 6 preforming line jog push-button [-366S1|E077.0]
   DB91_DBX085_2 : BOOL ;
   DB91_DBX085_3 : BOOL ;
   DB91_DBX085_4 : BOOL ;
   DB91_DBX085_5 : BOOL ;
   DB91_DBX085_6 : BOOL ;
   DB91_DBX085_7 : BOOL ;
   DB91_DBX086_0 : BOOL ;
   DB91_DBX086_1 : BOOL ;
   DB91_DBX086_2 : BOOL ;
   DB91_DBX086_3 : BOOL ;
   DB91_DBX086_4 : BOOL ;
   DB91_DBX086_5 : BOOL ;
   DB91_DBX086_6 : BOOL ;
   DB91_DBX086_7 : BOOL ;
   DB91_DBX087_0 : BOOL ;	//Cage 6 bobbin brakes air tank minimum pressure pressure-switch [-367S7|E077.7]
   DB91_DBX087_1 : BOOL ;	//Cage 6 line 1 pintles open [-367S8|E078.0]
   DB91_DBX087_2 : BOOL ;	//Cage 6 line 2 pintles open [-368S1|E078.1]
   DB91_DBX087_3 : BOOL ;	//Cage 6 line 3 pintles open [-368S2|E078.2]
   DB91_DBX087_4 : BOOL ;
   DB91_DBX087_5 : BOOL ;
   DB91_DBX087_6 : BOOL ;
   DB91_DBX087_7 : BOOL ;
   DB91_DBX088_0 : BOOL ;
   DB91_DBX088_1 : BOOL ;
   DB91_DBX088_2 : BOOL ;
   DB91_DBX088_3 : BOOL ;
   DB91_DBX088_4 : BOOL ;
   DB91_DBX088_5 : BOOL ;
   DB91_DBX088_6 : BOOL ;
   DB91_DBX088_7 : BOOL ;
   DB91_DBX089_0 : BOOL ;
   DB91_DBX089_1 : BOOL ;
   DB91_DBX089_2 : BOOL ;
   DB91_DBX089_3 : BOOL ;
   DB91_DBX089_4 : BOOL ;
   DB91_DBX089_5 : BOOL ;
   DB91_DBX089_6 : BOOL ;
   DB91_DBX089_7 : BOOL ;
   DB91_DBX090_0 : BOOL ;	//Cage 6 bobbin 1 break of wire and diameter calculation [-367B1|E077.1]
   DB91_DBX090_1 : BOOL ;	//Cage 6 bobbin 2 break of wire [-367B2|E077.2]
   DB91_DBX090_2 : BOOL ;	//Cage 6 bobbin 3 break of wire [-367B3|E077.3]
   DB91_DBX090_3 : BOOL ;	//Cage 6 bobbin 4 break of wire [-367B4|E077.4]
   DB91_DBX090_4 : BOOL ;	//Cage 6 bobbin 5 break of wire [-367B5|E077.5]
   DB91_DBX090_5 : BOOL ;	//Cage 6 bobbin 6 break of wire [-367B6|E077.6]
   DB91_DBX090_6 : BOOL ;
   DB91_DBX090_7 : BOOL ;
   DB91_DBX091_0 : BOOL ;
   DB91_DBX091_1 : BOOL ;
   DB91_DBX091_2 : BOOL ;
   DB91_DBX091_3 : BOOL ;
   DB91_DBX091_4 : BOOL ;
   DB91_DBX091_5 : BOOL ;
   DB91_DBX091_6 : BOOL ;
   DB91_DBX091_7 : BOOL ;
   DB91_DBX092_0 : BOOL ;
   DB91_DBX092_1 : BOOL ;
   DB91_DBX092_2 : BOOL ;
   DB91_DBX092_3 : BOOL ;
   DB91_DBX092_4 : BOOL ;
   DB91_DBX092_5 : BOOL ;
   DB91_DBX092_6 : BOOL ;
   DB91_DBX092_7 : BOOL ;
   DB91_DBX093_0 : BOOL ;
   DB91_DBX093_1 : BOOL ;
   DB91_DBX093_2 : BOOL ;
   DB91_DBX093_3 : BOOL ;
   DB91_DBX093_4 : BOOL ;
   DB91_DBX093_5 : BOOL ;
   DB91_DBX093_6 : BOOL ;
   DB91_DBX093_7 : BOOL ;
   DB91_DBX094_0 : BOOL ;
   DB91_DBX094_1 : BOOL ;
   DB91_DBX094_2 : BOOL ;
   DB91_DBX094_3 : BOOL ;
   DB91_DBX094_4 : BOOL ;
   DB91_DBX094_5 : BOOL ;
   DB91_DBX094_6 : BOOL ;
   DB91_DBX094_7 : BOOL ;
   DB91_DBX095_0 : BOOL ;
   DB91_DBX095_1 : BOOL ;
   DB91_DBX095_2 : BOOL ;
   DB91_DBX095_3 : BOOL ;
   DB91_DBX095_4 : BOOL ;
   DB91_DBX095_5 : BOOL ;
   DB91_DBX095_6 : BOOL ;
   DB91_DBX095_7 : BOOL ;
   DB91_DBX096_0 : BOOL ;	//Cage 6 Loader in stand by zone [+MCB06:7|E009.0]
   DB91_DBX096_1 : BOOL ;	//Cage 6 Loader inside cage [+MCB06:8|E009.1]
   DB91_DBX096_2 : BOOL ;	//Cage 6 Loader open clamp [+MCB06:9|E009.2]
   DB91_DBX096_3 : BOOL ;	//Cage 6 Loader to parcking zone [+MCB06:10|E009.3]
   DB91_DBX096_4 : BOOL ;
   DB91_DBX096_5 : BOOL ;
   DB91_DBX096_6 : BOOL ;
   DB91_DBX096_7 : BOOL ;
   DB91_DBX097_0 : BOOL ;	//Cage 6 loader locked
   DB91_DBX097_1 : BOOL ;	//Cage 6 loader unlocked
   DB91_DBX097_2 : BOOL ;
   DB91_DBX097_3 : BOOL ;
   DB91_DBX097_4 : BOOL ;
   DB91_DBX097_5 : BOOL ;
   DB91_DBX097_6 : BOOL ;
   DB91_DBX097_7 : BOOL ;
   DB91_DBX098_0 : BOOL ;
   DB91_DBX098_1 : BOOL ;
   DB91_DBX098_2 : BOOL ;
   DB91_DBX098_3 : BOOL ;
   DB91_DBX098_4 : BOOL ;
   DB91_DBX098_5 : BOOL ;
   DB91_DBX098_6 : BOOL ;
   DB91_DBX098_7 : BOOL ;
   DB91_DBX099_0 : BOOL ;	//Central Pay-off 630 pintle close selector-switch [-375S1|E078.7]
   DB91_DBX099_1 : BOOL ;	//Central Pay-off 630 break of wire sensor [-375B1|E079.0]
   DB91_DBX099_2 : BOOL ;	//Central Pay-off 630 main air minimum pressure-switch [-375S3|E079.1]
   DB91_DBX099_3 : BOOL ;	//Central Pay-off 630 line stop push-button [-375S4|E079.2]
   DB91_DBX099_4 : BOOL ;	//Central Pay-off 630 break release push-button [-375S5|E079.3]
   DB91_DBX099_5 : BOOL ;
   DB91_DBX099_6 : BOOL ;
   DB91_DBX099_7 : BOOL ;
   DB91_DBX100_0 : BOOL ;
   DB91_DBX100_1 : BOOL ;
   DB91_DBX100_2 : BOOL ;
   DB91_DBX100_3 : BOOL ;
   DB91_DBX100_4 : BOOL ;
   DB91_DBX100_5 : BOOL ;
   DB91_DBX100_6 : BOOL ;
   DB91_DBX100_7 : BOOL ;
   DB91_DBX101_0 : BOOL ;
   DB91_DBX101_1 : BOOL ;
   DB91_DBX101_2 : BOOL ;
   DB91_DBX101_3 : BOOL ;
   DB91_DBX101_4 : BOOL ;
   DB91_DBX101_5 : BOOL ;
   DB91_DBX101_6 : BOOL ;
   DB91_DBX101_7 : BOOL ;
   DB91_DBX102_0 : BOOL ;
   DB91_DBX102_1 : BOOL ;
   DB91_DBX102_2 : BOOL ;
   DB91_DBX102_3 : BOOL ;
   DB91_DBX102_4 : BOOL ;
   DB91_DBX102_5 : BOOL ;
   DB91_DBX102_6 : BOOL ;
   DB91_DBX102_7 : BOOL ;
   DB91_DBX103_0 : BOOL ;
   DB91_DBX103_1 : BOOL ;
   DB91_DBX103_2 : BOOL ;
   DB91_DBX103_3 : BOOL ;
   DB91_DBX103_4 : BOOL ;
   DB91_DBX103_5 : BOOL ;
   DB91_DBX103_6 : BOOL ;
   DB91_DBX103_7 : BOOL ;
   DB91_DBX104_0 : BOOL ;
   DB91_DBX104_1 : BOOL ;
   DB91_DBX104_2 : BOOL ;
   DB91_DBX104_3 : BOOL ;
   DB91_DBX104_4 : BOOL ;
   DB91_DBX104_5 : BOOL ;
   DB91_DBX104_6 : BOOL ;
   DB91_DBX104_7 : BOOL ;
   DB91_DBX105_0 : BOOL ;
   DB91_DBX105_1 : BOOL ;
   DB91_DBX105_2 : BOOL ;
   DB91_DBX105_3 : BOOL ;
   DB91_DBX105_4 : BOOL ;
   DB91_DBX105_5 : BOOL ;
   DB91_DBX105_6 : BOOL ;
   DB91_DBX105_7 : BOOL ;
   DB91_DBX106_0 : BOOL ;
   DB91_DBX106_1 : BOOL ;
   DB91_DBX106_2 : BOOL ;
   DB91_DBX106_3 : BOOL ;
   DB91_DBX106_4 : BOOL ;
   DB91_DBX106_5 : BOOL ;
   DB91_DBX106_6 : BOOL ;
   DB91_DBX106_7 : BOOL ;
   DB91_DBX107_0 : BOOL ;
   DB91_DBX107_1 : BOOL ;
   DB91_DBX107_2 : BOOL ;
   DB91_DBX107_3 : BOOL ;
   DB91_DBX107_4 : BOOL ;
   DB91_DBX107_5 : BOOL ;
   DB91_DBX107_6 : BOOL ;
   DB91_DBX107_7 : BOOL ;
   DB91_DBX108_0 : BOOL ;
   DB91_DBX108_1 : BOOL ;
   DB91_DBX108_2 : BOOL ;
   DB91_DBX108_3 : BOOL ;
   DB91_DBX108_4 : BOOL ;
   DB91_DBX108_5 : BOOL ;
   DB91_DBX108_6 : BOOL ;
   DB91_DBX108_7 : BOOL ;
   DB91_DBX109_0 : BOOL ;
   DB91_DBX109_1 : BOOL ;
   DB91_DBX109_2 : BOOL ;
   DB91_DBX109_3 : BOOL ;
   DB91_DBX109_4 : BOOL ;
   DB91_DBX109_5 : BOOL ;
   DB91_DBX109_6 : BOOL ;
   DB91_DBX109_7 : BOOL ;
   DB91_DBX110_0 : BOOL ;
   DB91_DBX110_1 : BOOL ;
   DB91_DBX110_2 : BOOL ;
   DB91_DBX110_3 : BOOL ;
   DB91_DBX110_4 : BOOL ;
   DB91_DBX110_5 : BOOL ;
   DB91_DBX110_6 : BOOL ;
   DB91_DBX110_7 : BOOL ;
   DB91_DBX111_0 : BOOL ;
   DB91_DBX111_1 : BOOL ;
   DB91_DBX111_2 : BOOL ;
   DB91_DBX111_3 : BOOL ;
   DB91_DBX111_4 : BOOL ;
   DB91_DBX111_5 : BOOL ;
   DB91_DBX111_6 : BOOL ;
   DB91_DBX111_7 : BOOL ;
   DB91_DBX112_0 : BOOL ;
   DB91_DBX112_1 : BOOL ;
   DB91_DBX112_2 : BOOL ;
   DB91_DBX112_3 : BOOL ;
   DB91_DBX112_4 : BOOL ;
   DB91_DBX112_5 : BOOL ;
   DB91_DBX112_6 : BOOL ;
   DB91_DBX112_7 : BOOL ;
   DB91_DBX113_0 : BOOL ;
   DB91_DBX113_1 : BOOL ;
   DB91_DBX113_2 : BOOL ;
   DB91_DBX113_3 : BOOL ;
   DB91_DBX113_4 : BOOL ;
   DB91_DBX113_5 : BOOL ;
   DB91_DBX113_6 : BOOL ;
   DB91_DBX113_7 : BOOL ;
   DB91_DBX114_0 : BOOL ;
   DB91_DBX114_1 : BOOL ;
   DB91_DBX114_2 : BOOL ;
   DB91_DBX114_3 : BOOL ;
   DB91_DBX114_4 : BOOL ;
   DB91_DBX114_5 : BOOL ;
   DB91_DBX114_6 : BOOL ;
   DB91_DBX114_7 : BOOL ;
   DB91_DBX115_0 : BOOL ;
   DB91_DBX115_1 : BOOL ;
   DB91_DBX115_2 : BOOL ;
   DB91_DBX115_3 : BOOL ;
   DB91_DBX115_4 : BOOL ;
   DB91_DBX115_5 : BOOL ;
   DB91_DBX115_6 : BOOL ;
   DB91_DBX115_7 : BOOL ;
   DB91_DBX116_0 : BOOL ;
   DB91_DBX116_1 : BOOL ;
   DB91_DBX116_2 : BOOL ;
   DB91_DBX116_3 : BOOL ;
   DB91_DBX116_4 : BOOL ;
   DB91_DBX116_5 : BOOL ;
   DB91_DBX116_6 : BOOL ;
   DB91_DBX116_7 : BOOL ;
   DB91_DBX117_0 : BOOL ;
   DB91_DBX117_1 : BOOL ;
   DB91_DBX117_2 : BOOL ;
   DB91_DBX117_3 : BOOL ;
   DB91_DBX117_4 : BOOL ;
   DB91_DBX117_5 : BOOL ;
   DB91_DBX117_6 : BOOL ;
   DB91_DBX117_7 : BOOL ;
   DB91_DBX118_0 : BOOL ;
   DB91_DBX118_1 : BOOL ;
   DB91_DBX118_2 : BOOL ;
   DB91_DBX118_3 : BOOL ;
   DB91_DBX118_4 : BOOL ;
   DB91_DBX118_5 : BOOL ;
   DB91_DBX118_6 : BOOL ;
   DB91_DBX118_7 : BOOL ;
   DB91_DBX119_0 : BOOL ;
   DB91_DBX119_1 : BOOL ;
   DB91_DBX119_2 : BOOL ;
   DB91_DBX119_3 : BOOL ;
   DB91_DBX119_4 : BOOL ;
   DB91_DBX119_5 : BOOL ;
   DB91_DBX119_6 : BOOL ;
   DB91_DBX119_7 : BOOL ;
   DB91_DBX120_0 : BOOL ;
   DB91_DBX120_1 : BOOL ;
   DB91_DBX120_2 : BOOL ;
   DB91_DBX120_3 : BOOL ;
   DB91_DBX120_4 : BOOL ;
   DB91_DBX120_5 : BOOL ;
   DB91_DBX120_6 : BOOL ;
   DB91_DBX120_7 : BOOL ;
   DB91_DBX121_0 : BOOL ;
   DB91_DBX121_1 : BOOL ;
   DB91_DBX121_2 : BOOL ;
   DB91_DBX121_3 : BOOL ;
   DB91_DBX121_4 : BOOL ;
   DB91_DBX121_5 : BOOL ;
   DB91_DBX121_6 : BOOL ;
   DB91_DBX121_7 : BOOL ;
   DB91_DBX122_0 : BOOL ;
   DB91_DBX122_1 : BOOL ;
   DB91_DBX122_2 : BOOL ;
   DB91_DBX122_3 : BOOL ;
   DB91_DBX122_4 : BOOL ;
   DB91_DBX122_5 : BOOL ;
   DB91_DBX122_6 : BOOL ;
   DB91_DBX122_7 : BOOL ;
   DB91_DBX123_0 : BOOL ;
   DB91_DBX123_1 : BOOL ;
   DB91_DBX123_2 : BOOL ;
   DB91_DBX123_3 : BOOL ;
   DB91_DBX123_4 : BOOL ;
   DB91_DBX123_5 : BOOL ;
   DB91_DBX123_6 : BOOL ;
   DB91_DBX123_7 : BOOL ;
   DB91_DBX124_0 : BOOL ;
   DB91_DBX124_1 : BOOL ;
   DB91_DBX124_2 : BOOL ;
   DB91_DBX124_3 : BOOL ;
   DB91_DBX124_4 : BOOL ;
   DB91_DBX124_5 : BOOL ;
   DB91_DBX124_6 : BOOL ;
   DB91_DBX124_7 : BOOL ;
   DB91_DBX125_0 : BOOL ;
   DB91_DBX125_1 : BOOL ;
   DB91_DBX125_2 : BOOL ;
   DB91_DBX125_3 : BOOL ;
   DB91_DBX125_4 : BOOL ;
   DB91_DBX125_5 : BOOL ;
   DB91_DBX125_6 : BOOL ;
   DB91_DBX125_7 : BOOL ;
   DB91_DBX126_0 : BOOL ;
   DB91_DBX126_1 : BOOL ;
   DB91_DBX126_2 : BOOL ;
   DB91_DBX126_3 : BOOL ;
   DB91_DBX126_4 : BOOL ;
   DB91_DBX126_5 : BOOL ;
   DB91_DBX126_6 : BOOL ;
   DB91_DBX126_7 : BOOL ;
   DB91_DBX127_0 : BOOL ;
   DB91_DBX127_1 : BOOL ;
   DB91_DBX127_2 : BOOL ;
   DB91_DBX127_3 : BOOL ;
   DB91_DBX127_4 : BOOL ;
   DB91_DBX127_5 : BOOL ;
   DB91_DBX127_6 : BOOL ;
   DB91_DBX127_7 : BOOL ;
   DB91_DBX128_0 : BOOL ;
   DB91_DBX128_1 : BOOL ;
   DB91_DBX128_2 : BOOL ;
   DB91_DBX128_3 : BOOL ;
   DB91_DBX128_4 : BOOL ;
   DB91_DBX128_5 : BOOL ;
   DB91_DBX128_6 : BOOL ;
   DB91_DBX128_7 : BOOL ;
   DB91_DBX129_0 : BOOL ;
   DB91_DBX129_1 : BOOL ;
   DB91_DBX129_2 : BOOL ;
   DB91_DBX129_3 : BOOL ;
   DB91_DBX129_4 : BOOL ;
   DB91_DBX129_5 : BOOL ;
   DB91_DBX129_6 : BOOL ;
   DB91_DBX129_7 : BOOL ;
   DB91_DBX130_0 : BOOL ;
   DB91_DBX130_1 : BOOL ;
   DB91_DBX130_2 : BOOL ;
   DB91_DBX130_3 : BOOL ;
   DB91_DBX130_4 : BOOL ;
   DB91_DBX130_5 : BOOL ;
   DB91_DBX130_6 : BOOL ;
   DB91_DBX130_7 : BOOL ;
   DB91_DBX131_0 : BOOL ;
   DB91_DBX131_1 : BOOL ;
   DB91_DBX131_2 : BOOL ;
   DB91_DBX131_3 : BOOL ;
   DB91_DBX131_4 : BOOL ;
   DB91_DBX131_5 : BOOL ;
   DB91_DBX131_6 : BOOL ;
   DB91_DBX131_7 : BOOL ;
   DB91_DBX132_0 : BOOL ;
   DB91_DBX132_1 : BOOL ;
   DB91_DBX132_2 : BOOL ;
   DB91_DBX132_3 : BOOL ;
   DB91_DBX132_4 : BOOL ;
   DB91_DBX132_5 : BOOL ;
   DB91_DBX132_6 : BOOL ;
   DB91_DBX132_7 : BOOL ;
   DB91_DBX133_0 : BOOL ;
   DB91_DBX133_1 : BOOL ;
   DB91_DBX133_2 : BOOL ;
   DB91_DBX133_3 : BOOL ;
   DB91_DBX133_4 : BOOL ;
   DB91_DBX133_5 : BOOL ;
   DB91_DBX133_6 : BOOL ;
   DB91_DBX133_7 : BOOL ;
   DB91_DBX134_0 : BOOL ;
   DB91_DBX134_1 : BOOL ;
   DB91_DBX134_2 : BOOL ;
   DB91_DBX134_3 : BOOL ;
   DB91_DBX134_4 : BOOL ;
   DB91_DBX134_5 : BOOL ;
   DB91_DBX134_6 : BOOL ;
   DB91_DBX134_7 : BOOL ;
   DB91_DBX135_0 : BOOL ;
   DB91_DBX135_1 : BOOL ;
   DB91_DBX135_2 : BOOL ;
   DB91_DBX135_3 : BOOL ;
   DB91_DBX135_4 : BOOL ;
   DB91_DBX135_5 : BOOL ;
   DB91_DBX135_6 : BOOL ;
   DB91_DBX135_7 : BOOL ;
   DB91_DBX136_0 : BOOL ;
   DB91_DBX136_1 : BOOL ;
   DB91_DBX136_2 : BOOL ;
   DB91_DBX136_3 : BOOL ;
   DB91_DBX136_4 : BOOL ;
   DB91_DBX136_5 : BOOL ;
   DB91_DBX136_6 : BOOL ;
   DB91_DBX136_7 : BOOL ;
   DB91_DBX137_0 : BOOL ;
   DB91_DBX137_1 : BOOL ;
   DB91_DBX137_2 : BOOL ;
   DB91_DBX137_3 : BOOL ;
   DB91_DBX137_4 : BOOL ;
   DB91_DBX137_5 : BOOL ;
   DB91_DBX137_6 : BOOL ;
   DB91_DBX137_7 : BOOL ;
   DB91_DBX138_0 : BOOL ;
   DB91_DBX138_1 : BOOL ;
   DB91_DBX138_2 : BOOL ;
   DB91_DBX138_3 : BOOL ;
   DB91_DBX138_4 : BOOL ;
   DB91_DBX138_5 : BOOL ;
   DB91_DBX138_6 : BOOL ;
   DB91_DBX138_7 : BOOL ;
   DB91_DBX139_0 : BOOL ;
   DB91_DBX139_1 : BOOL ;
   DB91_DBX139_2 : BOOL ;
   DB91_DBX139_3 : BOOL ;
   DB91_DBX139_4 : BOOL ;
   DB91_DBX139_5 : BOOL ;
   DB91_DBX139_6 : BOOL ;
   DB91_DBX139_7 : BOOL ;
   DB91_DBX140_0 : BOOL ;
   DB91_DBX140_1 : BOOL ;
   DB91_DBX140_2 : BOOL ;
   DB91_DBX140_3 : BOOL ;
   DB91_DBX140_4 : BOOL ;
   DB91_DBX140_5 : BOOL ;
   DB91_DBX140_6 : BOOL ;
   DB91_DBX140_7 : BOOL ;
   DB91_DBX141_0 : BOOL ;
   DB91_DBX141_1 : BOOL ;
   DB91_DBX141_2 : BOOL ;
   DB91_DBX141_3 : BOOL ;
   DB91_DBX141_4 : BOOL ;
   DB91_DBX141_5 : BOOL ;
   DB91_DBX141_6 : BOOL ;
   DB91_DBX141_7 : BOOL ;
   DB91_DBX142_0 : BOOL ;
   DB91_DBX142_1 : BOOL ;
   DB91_DBX142_2 : BOOL ;
   DB91_DBX142_3 : BOOL ;
   DB91_DBX142_4 : BOOL ;
   DB91_DBX142_5 : BOOL ;
   DB91_DBX142_6 : BOOL ;
   DB91_DBX142_7 : BOOL ;
   DB91_DBX143_0 : BOOL ;
   DB91_DBX143_1 : BOOL ;
   DB91_DBX143_2 : BOOL ;
   DB91_DBX143_3 : BOOL ;
   DB91_DBX143_4 : BOOL ;
   DB91_DBX143_5 : BOOL ;
   DB91_DBX143_6 : BOOL ;
   DB91_DBX143_7 : BOOL ;
   DB91_DBX144_0 : BOOL ;
   DB91_DBX144_1 : BOOL ;
   DB91_DBX144_2 : BOOL ;
   DB91_DBX144_3 : BOOL ;
   DB91_DBX144_4 : BOOL ;
   DB91_DBX144_5 : BOOL ;
   DB91_DBX144_6 : BOOL ;
   DB91_DBX144_7 : BOOL ;
   DB91_DBX145_0 : BOOL ;
   DB91_DBX145_1 : BOOL ;
   DB91_DBX145_2 : BOOL ;
   DB91_DBX145_3 : BOOL ;
   DB91_DBX145_4 : BOOL ;
   DB91_DBX145_5 : BOOL ;
   DB91_DBX145_6 : BOOL ;
   DB91_DBX145_7 : BOOL ;
   DB91_DBX146_0 : BOOL ;
   DB91_DBX146_1 : BOOL ;
   DB91_DBX146_2 : BOOL ;
   DB91_DBX146_3 : BOOL ;
   DB91_DBX146_4 : BOOL ;
   DB91_DBX146_5 : BOOL ;
   DB91_DBX146_6 : BOOL ;
   DB91_DBX146_7 : BOOL ;
   DB91_DBX147_0 : BOOL ;
   DB91_DBX147_1 : BOOL ;
   DB91_DBX147_2 : BOOL ;
   DB91_DBX147_3 : BOOL ;
   DB91_DBX147_4 : BOOL ;
   DB91_DBX147_5 : BOOL ;
   DB91_DBX147_6 : BOOL ;
   DB91_DBX147_7 : BOOL ;
   DB91_DBX148_0 : BOOL ;
   DB91_DBX148_1 : BOOL ;
   DB91_DBX148_2 : BOOL ;
   DB91_DBX148_3 : BOOL ;
   DB91_DBX148_4 : BOOL ;
   DB91_DBX148_5 : BOOL ;
   DB91_DBX148_6 : BOOL ;
   DB91_DBX148_7 : BOOL ;
   DB91_DBX149_0 : BOOL ;
   DB91_DBX149_1 : BOOL ;
   DB91_DBX149_2 : BOOL ;
   DB91_DBX149_3 : BOOL ;
   DB91_DBX149_4 : BOOL ;
   DB91_DBX149_5 : BOOL ;
   DB91_DBX149_6 : BOOL ;
   DB91_DBX149_7 : BOOL ;
   DB91_DBX150_0 : BOOL ;
   DB91_DBX150_1 : BOOL ;
   DB91_DBX150_2 : BOOL ;
   DB91_DBX150_3 : BOOL ;
   DB91_DBX150_4 : BOOL ;
   DB91_DBX150_5 : BOOL ;
   DB91_DBX150_6 : BOOL ;
   DB91_DBX150_7 : BOOL ;
   DB91_DBX151_0 : BOOL ;
   DB91_DBX151_1 : BOOL ;
   DB91_DBX151_2 : BOOL ;
   DB91_DBX151_3 : BOOL ;
   DB91_DBX151_4 : BOOL ;
   DB91_DBX151_5 : BOOL ;
   DB91_DBX151_6 : BOOL ;
   DB91_DBX151_7 : BOOL ;
   DB91_DBX152_0 : BOOL ;
   DB91_DBX152_1 : BOOL ;
   DB91_DBX152_2 : BOOL ;
   DB91_DBX152_3 : BOOL ;
   DB91_DBX152_4 : BOOL ;
   DB91_DBX152_5 : BOOL ;
   DB91_DBX152_6 : BOOL ;
   DB91_DBX152_7 : BOOL ;
   DB91_DBX153_0 : BOOL ;
   DB91_DBX153_1 : BOOL ;
   DB91_DBX153_2 : BOOL ;
   DB91_DBX153_3 : BOOL ;
   DB91_DBX153_4 : BOOL ;
   DB91_DBX153_5 : BOOL ;
   DB91_DBX153_6 : BOOL ;
   DB91_DBX153_7 : BOOL ;
   DB91_DBX154_0 : BOOL ;
   DB91_DBX154_1 : BOOL ;
   DB91_DBX154_2 : BOOL ;
   DB91_DBX154_3 : BOOL ;
   DB91_DBX154_4 : BOOL ;
   DB91_DBX154_5 : BOOL ;
   DB91_DBX154_6 : BOOL ;
   DB91_DBX154_7 : BOOL ;
   DB91_DBX155_0 : BOOL ;
   DB91_DBX155_1 : BOOL ;
   DB91_DBX155_2 : BOOL ;
   DB91_DBX155_3 : BOOL ;
   DB91_DBX155_4 : BOOL ;
   DB91_DBX155_5 : BOOL ;
   DB91_DBX155_6 : BOOL ;
   DB91_DBX155_7 : BOOL ;
   DB91_DBX156_0 : BOOL ;
   DB91_DBX156_1 : BOOL ;
   DB91_DBX156_2 : BOOL ;
   DB91_DBX156_3 : BOOL ;
   DB91_DBX156_4 : BOOL ;
   DB91_DBX156_5 : BOOL ;
   DB91_DBX156_6 : BOOL ;
   DB91_DBX156_7 : BOOL ;
   DB91_DBX157_0 : BOOL ;
   DB91_DBX157_1 : BOOL ;
   DB91_DBX157_2 : BOOL ;
   DB91_DBX157_3 : BOOL ;
   DB91_DBX157_4 : BOOL ;
   DB91_DBX157_5 : BOOL ;
   DB91_DBX157_6 : BOOL ;
   DB91_DBX157_7 : BOOL ;
   DB91_DBX158_0 : BOOL ;
   DB91_DBX158_1 : BOOL ;
   DB91_DBX158_2 : BOOL ;
   DB91_DBX158_3 : BOOL ;
   DB91_DBX158_4 : BOOL ;
   DB91_DBX158_5 : BOOL ;
   DB91_DBX158_6 : BOOL ;
   DB91_DBX158_7 : BOOL ;
   DB91_DBX159_0 : BOOL ;
   DB91_DBX159_1 : BOOL ;
   DB91_DBX159_2 : BOOL ;
   DB91_DBX159_3 : BOOL ;
   DB91_DBX159_4 : BOOL ;
   DB91_DBX159_5 : BOOL ;
   DB91_DBX159_6 : BOOL ;
   DB91_DBX159_7 : BOOL ;
   DB91_DBX160_0 : BOOL ;
   DB91_DBX160_1 : BOOL ;
   DB91_DBX160_2 : BOOL ;
   DB91_DBX160_3 : BOOL ;
   DB91_DBX160_4 : BOOL ;
   DB91_DBX160_5 : BOOL ;
   DB91_DBX160_6 : BOOL ;
   DB91_DBX160_7 : BOOL ;
   DB91_DBX161_0 : BOOL ;
   DB91_DBX161_1 : BOOL ;
   DB91_DBX161_2 : BOOL ;
   DB91_DBX161_3 : BOOL ;
   DB91_DBX161_4 : BOOL ;
   DB91_DBX161_5 : BOOL ;
   DB91_DBX161_6 : BOOL ;
   DB91_DBX161_7 : BOOL ;
   DB91_DBX162_0 : BOOL ;
   DB91_DBX162_1 : BOOL ;
   DB91_DBX162_2 : BOOL ;
   DB91_DBX162_3 : BOOL ;
   DB91_DBX162_4 : BOOL ;
   DB91_DBX162_5 : BOOL ;
   DB91_DBX162_6 : BOOL ;
   DB91_DBX162_7 : BOOL ;
   DB91_DBX163_0 : BOOL ;
   DB91_DBX163_1 : BOOL ;
   DB91_DBX163_2 : BOOL ;
   DB91_DBX163_3 : BOOL ;
   DB91_DBX163_4 : BOOL ;
   DB91_DBX163_5 : BOOL ;
   DB91_DBX163_6 : BOOL ;
   DB91_DBX163_7 : BOOL ;
   DB91_DBX164_0 : BOOL ;
   DB91_DBX164_1 : BOOL ;
   DB91_DBX164_2 : BOOL ;
   DB91_DBX164_3 : BOOL ;
   DB91_DBX164_4 : BOOL ;
   DB91_DBX164_5 : BOOL ;
   DB91_DBX164_6 : BOOL ;
   DB91_DBX164_7 : BOOL ;
   DB91_DBX165_0 : BOOL ;
   DB91_DBX165_1 : BOOL ;
   DB91_DBX165_2 : BOOL ;
   DB91_DBX165_3 : BOOL ;
   DB91_DBX165_4 : BOOL ;
   DB91_DBX165_5 : BOOL ;
   DB91_DBX165_6 : BOOL ;
   DB91_DBX165_7 : BOOL ;
   DB91_DBX166_0 : BOOL ;
   DB91_DBX166_1 : BOOL ;
   DB91_DBX166_2 : BOOL ;
   DB91_DBX166_3 : BOOL ;
   DB91_DBX166_4 : BOOL ;
   DB91_DBX166_5 : BOOL ;
   DB91_DBX166_6 : BOOL ;
   DB91_DBX166_7 : BOOL ;
   DB91_DBX167_0 : BOOL ;
   DB91_DBX167_1 : BOOL ;
   DB91_DBX167_2 : BOOL ;
   DB91_DBX167_3 : BOOL ;
   DB91_DBX167_4 : BOOL ;
   DB91_DBX167_5 : BOOL ;
   DB91_DBX167_6 : BOOL ;
   DB91_DBX167_7 : BOOL ;
   DB91_DBX168_0 : BOOL ;
   DB91_DBX168_1 : BOOL ;
   DB91_DBX168_2 : BOOL ;
   DB91_DBX168_3 : BOOL ;
   DB91_DBX168_4 : BOOL ;
   DB91_DBX168_5 : BOOL ;
   DB91_DBX168_6 : BOOL ;
   DB91_DBX168_7 : BOOL ;
   DB91_DBX169_0 : BOOL ;
   DB91_DBX169_1 : BOOL ;
   DB91_DBX169_2 : BOOL ;
   DB91_DBX169_3 : BOOL ;
   DB91_DBX169_4 : BOOL ;
   DB91_DBX169_5 : BOOL ;
   DB91_DBX169_6 : BOOL ;
   DB91_DBX169_7 : BOOL ;
   DB91_DBX170_0 : BOOL ;
   DB91_DBX170_1 : BOOL ;
   DB91_DBX170_2 : BOOL ;
   DB91_DBX170_3 : BOOL ;
   DB91_DBX170_4 : BOOL ;
   DB91_DBX170_5 : BOOL ;
   DB91_DBX170_6 : BOOL ;
   DB91_DBX170_7 : BOOL ;
   DB91_DBX171_0 : BOOL ;
   DB91_DBX171_1 : BOOL ;
   DB91_DBX171_2 : BOOL ;
   DB91_DBX171_3 : BOOL ;
   DB91_DBX171_4 : BOOL ;
   DB91_DBX171_5 : BOOL ;
   DB91_DBX171_6 : BOOL ;
   DB91_DBX171_7 : BOOL ;
   DB91_DBX172_0 : BOOL ;
   DB91_DBX172_1 : BOOL ;
   DB91_DBX172_2 : BOOL ;
   DB91_DBX172_3 : BOOL ;
   DB91_DBX172_4 : BOOL ;
   DB91_DBX172_5 : BOOL ;
   DB91_DBX172_6 : BOOL ;
   DB91_DBX172_7 : BOOL ;
   DB91_DBX173_0 : BOOL ;
   DB91_DBX173_1 : BOOL ;
   DB91_DBX173_2 : BOOL ;
   DB91_DBX173_3 : BOOL ;
   DB91_DBX173_4 : BOOL ;
   DB91_DBX173_5 : BOOL ;
   DB91_DBX173_6 : BOOL ;
   DB91_DBX173_7 : BOOL ;
   DB91_DBX174_0 : BOOL ;
   DB91_DBX174_1 : BOOL ;
   DB91_DBX174_2 : BOOL ;
   DB91_DBX174_3 : BOOL ;
   DB91_DBX174_4 : BOOL ;
   DB91_DBX174_5 : BOOL ;
   DB91_DBX174_6 : BOOL ;
   DB91_DBX174_7 : BOOL ;
   DB91_DBX175_0 : BOOL ;
   DB91_DBX175_1 : BOOL ;
   DB91_DBX175_2 : BOOL ;
   DB91_DBX175_3 : BOOL ;
   DB91_DBX175_4 : BOOL ;
   DB91_DBX175_5 : BOOL ;
   DB91_DBX175_6 : BOOL ;
   DB91_DBX175_7 : BOOL ;
   DB91_DBX176_0 : BOOL ;
   DB91_DBX176_1 : BOOL ;
   DB91_DBX176_2 : BOOL ;
   DB91_DBX176_3 : BOOL ;
   DB91_DBX176_4 : BOOL ;
   DB91_DBX176_5 : BOOL ;
   DB91_DBX176_6 : BOOL ;
   DB91_DBX176_7 : BOOL ;
   DB91_DBX177_0 : BOOL ;
   DB91_DBX177_1 : BOOL ;
   DB91_DBX177_2 : BOOL ;
   DB91_DBX177_3 : BOOL ;
   DB91_DBX177_4 : BOOL ;
   DB91_DBX177_5 : BOOL ;
   DB91_DBX177_6 : BOOL ;
   DB91_DBX177_7 : BOOL ;
   DB91_DBX178_0 : BOOL ;
   DB91_DBX178_1 : BOOL ;
   DB91_DBX178_2 : BOOL ;
   DB91_DBX178_3 : BOOL ;
   DB91_DBX178_4 : BOOL ;
   DB91_DBX178_5 : BOOL ;
   DB91_DBX178_6 : BOOL ;
   DB91_DBX178_7 : BOOL ;
   DB91_DBX179_0 : BOOL ;
   DB91_DBX179_1 : BOOL ;
   DB91_DBX179_2 : BOOL ;
   DB91_DBX179_3 : BOOL ;
   DB91_DBX179_4 : BOOL ;
   DB91_DBX179_5 : BOOL ;
   DB91_DBX179_6 : BOOL ;
   DB91_DBX179_7 : BOOL ;
   DB91_DBX180_0 : BOOL ;
   DB91_DBX180_1 : BOOL ;
   DB91_DBX180_2 : BOOL ;
   DB91_DBX180_3 : BOOL ;
   DB91_DBX180_4 : BOOL ;
   DB91_DBX180_5 : BOOL ;
   DB91_DBX180_6 : BOOL ;
   DB91_DBX180_7 : BOOL ;
   DB91_DBX181_0 : BOOL ;
   DB91_DBX181_1 : BOOL ;
   DB91_DBX181_2 : BOOL ;
   DB91_DBX181_3 : BOOL ;
   DB91_DBX181_4 : BOOL ;
   DB91_DBX181_5 : BOOL ;
   DB91_DBX181_6 : BOOL ;
   DB91_DBX181_7 : BOOL ;
   DB91_DBX182_0 : BOOL ;
   DB91_DBX182_1 : BOOL ;
   DB91_DBX182_2 : BOOL ;
   DB91_DBX182_3 : BOOL ;
   DB91_DBX182_4 : BOOL ;
   DB91_DBX182_5 : BOOL ;
   DB91_DBX182_6 : BOOL ;
   DB91_DBX182_7 : BOOL ;
   DB91_DBX183_0 : BOOL ;
   DB91_DBX183_1 : BOOL ;
   DB91_DBX183_2 : BOOL ;
   DB91_DBX183_3 : BOOL ;
   DB91_DBX183_4 : BOOL ;
   DB91_DBX183_5 : BOOL ;
   DB91_DBX183_6 : BOOL ;
   DB91_DBX183_7 : BOOL ;
   DB91_DBX184_0 : BOOL ;
   DB91_DBX184_1 : BOOL ;
   DB91_DBX184_2 : BOOL ;
   DB91_DBX184_3 : BOOL ;
   DB91_DBX184_4 : BOOL ;
   DB91_DBX184_5 : BOOL ;
   DB91_DBX184_6 : BOOL ;
   DB91_DBX184_7 : BOOL ;
   DB91_DBX185_0 : BOOL ;
   DB91_DBX185_1 : BOOL ;
   DB91_DBX185_2 : BOOL ;
   DB91_DBX185_3 : BOOL ;
   DB91_DBX185_4 : BOOL ;
   DB91_DBX185_5 : BOOL ;
   DB91_DBX185_6 : BOOL ;
   DB91_DBX185_7 : BOOL ;
   DB91_DBX186_0 : BOOL ;
   DB91_DBX186_1 : BOOL ;
   DB91_DBX186_2 : BOOL ;
   DB91_DBX186_3 : BOOL ;
   DB91_DBX186_4 : BOOL ;
   DB91_DBX186_5 : BOOL ;
   DB91_DBX186_6 : BOOL ;
   DB91_DBX186_7 : BOOL ;
   DB91_DBX187_0 : BOOL ;
   DB91_DBX187_1 : BOOL ;
   DB91_DBX187_2 : BOOL ;
   DB91_DBX187_3 : BOOL ;
   DB91_DBX187_4 : BOOL ;
   DB91_DBX187_5 : BOOL ;
   DB91_DBX187_6 : BOOL ;
   DB91_DBX187_7 : BOOL ;
   DB91_DBX188_0 : BOOL ;
   DB91_DBX188_1 : BOOL ;
   DB91_DBX188_2 : BOOL ;
   DB91_DBX188_3 : BOOL ;
   DB91_DBX188_4 : BOOL ;
   DB91_DBX188_5 : BOOL ;
   DB91_DBX188_6 : BOOL ;
   DB91_DBX188_7 : BOOL ;
   DB91_DBX189_0 : BOOL ;
   DB91_DBX189_1 : BOOL ;
   DB91_DBX189_2 : BOOL ;
   DB91_DBX189_3 : BOOL ;
   DB91_DBX189_4 : BOOL ;
   DB91_DBX189_5 : BOOL ;
   DB91_DBX189_6 : BOOL ;
   DB91_DBX189_7 : BOOL ;
   DB91_DBX190_0 : BOOL ;
   DB91_DBX190_1 : BOOL ;
   DB91_DBX190_2 : BOOL ;
   DB91_DBX190_3 : BOOL ;
   DB91_DBX190_4 : BOOL ;
   DB91_DBX190_5 : BOOL ;
   DB91_DBX190_6 : BOOL ;
   DB91_DBX190_7 : BOOL ;
   DB91_DBX191_0 : BOOL ;
   DB91_DBX191_1 : BOOL ;
   DB91_DBX191_2 : BOOL ;
   DB91_DBX191_3 : BOOL ;
   DB91_DBX191_4 : BOOL ;
   DB91_DBX191_5 : BOOL ;
   DB91_DBX191_6 : BOOL ;
   DB91_DBX191_7 : BOOL ;
   DB91_DBX192_0 : BOOL ;
   DB91_DBX192_1 : BOOL ;
   DB91_DBX192_2 : BOOL ;
   DB91_DBX192_3 : BOOL ;
   DB91_DBX192_4 : BOOL ;
   DB91_DBX192_5 : BOOL ;
   DB91_DBX192_6 : BOOL ;
   DB91_DBX192_7 : BOOL ;
   DB91_DBX193_0 : BOOL ;
   DB91_DBX193_1 : BOOL ;
   DB91_DBX193_2 : BOOL ;
   DB91_DBX193_3 : BOOL ;
   DB91_DBX193_4 : BOOL ;
   DB91_DBX193_5 : BOOL ;
   DB91_DBX193_6 : BOOL ;
   DB91_DBX193_7 : BOOL ;
   DB91_DBX194_0 : BOOL ;
   DB91_DBX194_1 : BOOL ;
   DB91_DBX194_2 : BOOL ;
   DB91_DBX194_3 : BOOL ;
   DB91_DBX194_4 : BOOL ;
   DB91_DBX194_5 : BOOL ;
   DB91_DBX194_6 : BOOL ;
   DB91_DBX194_7 : BOOL ;
   DB91_DBX195_0 : BOOL ;
   DB91_DBX195_1 : BOOL ;
   DB91_DBX195_2 : BOOL ;
   DB91_DBX195_3 : BOOL ;
   DB91_DBX195_4 : BOOL ;
   DB91_DBX195_5 : BOOL ;
   DB91_DBX195_6 : BOOL ;
   DB91_DBX195_7 : BOOL ;
   DB91_DBX196_0 : BOOL ;
   DB91_DBX196_1 : BOOL ;
   DB91_DBX196_2 : BOOL ;
   DB91_DBX196_3 : BOOL ;
   DB91_DBX196_4 : BOOL ;
   DB91_DBX196_5 : BOOL ;
   DB91_DBX196_6 : BOOL ;
   DB91_DBX196_7 : BOOL ;
  END_STRUCT ;	
BEGIN
   DB91_DBX000_0 := TRUE;
   DB91_DBX000_1 := TRUE;
   DB91_DBX000_2 := TRUE;
   DB91_DBX000_3 := TRUE;
   DB91_DBX000_4 := TRUE;
   DB91_DBX000_5 := TRUE;
   DB91_DBX000_6 := TRUE;
   DB91_DBX001_0 := TRUE;
   DB91_DBX001_1 := TRUE;
   DB91_DBX001_2 := TRUE;
   DB91_DBX002_0 := TRUE;
   DB91_DBX002_5 := TRUE;
   DB91_DBX003_1 := TRUE;
   DB91_DBX003_2 := TRUE;
   DB91_DBX003_3 := TRUE;
   DB91_DBX003_4 := TRUE;
   DB91_DBX004_2 := TRUE;
   DB91_DBX006_0 := TRUE;
   DB91_DBX006_1 := TRUE;
   DB91_DBX006_2 := TRUE;
   DB91_DBX006_3 := TRUE;
   DB91_DBX007_4 := TRUE;
   DB91_DBX007_5 := TRUE;
   DB91_DBX008_4 := TRUE;
   DB91_DBX009_2 := TRUE;
   DB91_DBX009_3 := TRUE;
   DB91_DBX012_1 := TRUE;
   DB91_DBX018_0 := TRUE;
   DB91_DBX018_1 := TRUE;
   DB91_DBX020_0 := TRUE;
   DB91_DBX020_2 := TRUE;
   DB91_DBX020_3 := TRUE;
   DB91_DBX020_5 := TRUE;
   DB91_DBX020_7 := TRUE;
   DB91_DBX021_1 := TRUE;
   DB91_DBX021_2 := TRUE;
   DB91_DBX021_4 := TRUE;
   DB91_DBX021_7 := TRUE;
   DB91_DBX022_0 := TRUE;
   DB91_DBX025_0 := TRUE;
   DB91_DBX027_4 := TRUE;
   DB91_DBX027_5 := TRUE;
   DB91_DBX027_6 := TRUE;
   DB91_DBX027_7 := TRUE;
   DB91_DBX030_5 := TRUE;
   DB91_DBX032_0 := TRUE;
   DB91_DBX032_1 := TRUE;
   DB91_DBX032_2 := TRUE;
   DB91_DBX032_3 := TRUE;
   DB91_DBX032_4 := TRUE;
   DB91_DBX032_5 := TRUE;
   DB91_DBX038_0 := TRUE;
   DB91_DBX038_1 := TRUE;
   DB91_DBX040_0 := TRUE;
   DB91_DBX040_2 := TRUE;
   DB91_DBX040_3 := TRUE;
   DB91_DBX040_5 := TRUE;
   DB91_DBX040_7 := TRUE;
   DB91_DBX041_1 := TRUE;
   DB91_DBX041_2 := TRUE;
   DB91_DBX041_4 := TRUE;
   DB91_DBX041_7 := TRUE;
   DB91_DBX042_0 := TRUE;
   DB91_DBX045_0 := TRUE;
   DB91_DBX047_0 := TRUE;
   DB91_DBX047_1 := TRUE;
   DB91_DBX047_2 := TRUE;
   DB91_DBX047_3 := TRUE;
   DB91_DBX050_2 := TRUE;
   DB91_DBX050_4 := TRUE;
   DB91_DBX050_6 := TRUE;
   DB91_DBX050_7 := TRUE;
   DB91_DBX051_0 := TRUE;
   DB91_DBX051_6 := TRUE;
   DB91_DBX052_1 := TRUE;
   DB91_DBX056_3 := TRUE;
   DB91_DBX056_5 := TRUE;
   DB91_DBX058_0 := TRUE;
   DB91_DBX058_1 := TRUE;
   DB91_DBX060_2 := TRUE;
   DB91_DBX060_4 := TRUE;
   DB91_DBX060_6 := TRUE;
   DB91_DBX060_7 := TRUE;
   DB91_DBX061_2 := TRUE;
   DB91_DBX061_4 := TRUE;
   DB91_DBX061_5 := TRUE;
   DB91_DBX061_6 := TRUE;
   DB91_DBX061_7 := TRUE;
   DB91_DBX062_0 := TRUE;
   DB91_DBX065_0 := TRUE;
   DB91_DBX067_0 := TRUE;
   DB91_DBX067_1 := TRUE;
   DB91_DBX067_2 := TRUE;
   DB91_DBX067_3 := TRUE;
   DB91_DBX070_2 := TRUE;
   DB91_DBX070_5 := TRUE;
   DB91_DBX070_7 := TRUE;
   DB91_DBX071_0 := TRUE;
   DB91_DBX071_2 := TRUE;
   DB91_DBX076_3 := TRUE;
   DB91_DBX077_1 := TRUE;
   DB91_DBX078_2 := TRUE;
   DB91_DBX078_3 := TRUE;
   DB91_DBX080_2 := TRUE;
   DB91_DBX080_4 := TRUE;
   DB91_DBX080_6 := TRUE;
   DB91_DBX080_7 := TRUE;
   DB91_DBX081_2 := TRUE;
   DB91_DBX081_4 := TRUE;
   DB91_DBX081_5 := TRUE;
   DB91_DBX081_6 := TRUE;
   DB91_DBX081_7 := TRUE;
   DB91_DBX082_0 := TRUE;
   DB91_DBX084_6 := TRUE;
   DB91_DBX085_0 := TRUE;
   DB91_DBX087_0 := TRUE;
   DB91_DBX087_1 := TRUE;
   DB91_DBX087_2 := TRUE;
   DB91_DBX087_3 := TRUE;
   DB91_DBX090_3 := TRUE;
   DB91_DBX090_4 := TRUE;
   DB91_DBX090_5 := TRUE;
   DB91_DBX097_1 := TRUE;
   DB91_DBX099_0 := TRUE;
   DB91_DBX099_2 := TRUE;
   DB91_DBX099_3 := TRUE;
END_DATA_BLOCK

DATA_BLOCK "MAP_DO"	// DB 93
TITLE = Mappa Uscite
VERSION : 0.0
  STRUCT
   DB93_DBX000_0 : BOOL ;	//Line run pilot lamp [-177S2:LAMP|A003.2]
   DB93_DBX000_1 : BOOL ;	//Alarms reset pilot lamps [-183K2|A003.3]
   DB93_DBX000_2 : BOOL ;	//Hold line speed pilot lamp [-177S5:LAMP|A003.4]
   DB93_DBX000_3 : BOOL ;	//Line start siren [-183K4|A003.5]
   DB93_DBX000_4 : BOOL ;	//Drives feeder reset [-140G1:X101:10|A003.6]
   DB93_DBX000_5 : BOOL ;	//Breaking unit reset [-141A1:1|A003.7]
   DB93_DBX000_6 : BOOL ;	//Drives feeder start [-140G1:X101:9|A000.0]
   DB93_DBX000_7 : BOOL ;
   DB93_DBX001_0 : BOOL ;
   DB93_DBX001_1 : BOOL ;
   DB93_DBX001_2 : BOOL ;	//Capstan motor blower contactor [-732K1|A000.4]
   DB93_DBX001_3 : BOOL ;	//Capstan motor block brake electric valve [-732Y2|A000.5]
   DB93_DBX001_4 : BOOL ;	//Cable block opening electric valve [-732Y3|A000.6]
   DB93_DBX001_5 : BOOL ;
   DB93_DBX001_6 : BOOL ;
   DB93_DBX001_7 : BOOL ;
   DB93_DBX002_0 : BOOL ;	//230 VAC UPS automatic shut-down [-193K1|A005.0]
   DB93_DBX002_1 : BOOL ;
   DB93_DBX002_2 : BOOL ;
   DB93_DBX002_3 : BOOL ;
   DB93_DBX002_4 : BOOL ;
   DB93_DBX002_5 : BOOL ;
   DB93_DBX002_6 : BOOL ;
   DB93_DBX002_7 : BOOL ;
   DB93_DBX003_0 : BOOL ;
   DB93_DBX003_1 : BOOL ;
   DB93_DBX003_2 : BOOL ;
   DB93_DBX003_3 : BOOL ;
   DB93_DBX003_4 : BOOL ;
   DB93_DBX003_5 : BOOL ;
   DB93_DBX003_6 : BOOL ;
   DB93_DBX003_7 : BOOL ;
   DB93_DBX004_0 : BOOL ;	//Take-up idle pintle up motor contactor [-981K1|A032.0]
   DB93_DBX004_1 : BOOL ;	//Take-up idle pintle down motor contactor [-981K2|A032.1]
   DB93_DBX004_2 : BOOL ;	//Take-up driven pintle up motor contactor [-981K3|A032.2]
   DB93_DBX004_3 : BOOL ;	//Take-up driven pintle down motor contactor [-981K4|A032.3]
   DB93_DBX004_4 : BOOL ;	//Take-up idle pintle opening motor contactor [-981K5|A033.0]
   DB93_DBX004_5 : BOOL ;	//Take-up idle pintle closing motor contactor [-981K6|A033.1]
   DB93_DBX004_6 : BOOL ;	//Take-up traverse left direction pilot lamps [-981K7|A033.2]
   DB93_DBX004_7 : BOOL ;	//Take-up traverse right direction pilot lamps [-981K8|A033.3]
   DB93_DBX005_0 : BOOL ;	//Take-up traverse motor blower contactor [-982K1|A034.0]
   DB93_DBX005_1 : BOOL ;	//Take-up bobbin motor blower contactor [-982K2|A034.1]
   DB93_DBX005_2 : BOOL ;	//Take-up bobbin electric brake relay [-982K3|A034.2]
   DB93_DBX005_3 : BOOL ;
   DB93_DBX005_4 : BOOL ;
   DB93_DBX005_5 : BOOL ;
   DB93_DBX005_6 : BOOL ;
   DB93_DBX005_7 : BOOL ;
   DB93_DBX006_0 : BOOL ;	//Take-up traverse quick left pilot lamp [-922S3:LAMP|A000.1]
   DB93_DBX006_1 : BOOL ;	//Take-up traverse quick right pilot lamp [-922S4:LAMP|A000.2]
   DB93_DBX006_2 : BOOL ;	//Take-up bobbin run pilot lamps [-925K3|A000.3]
   DB93_DBX006_3 : BOOL ;
   DB93_DBX006_4 : BOOL ;
   DB93_DBX006_5 : BOOL ;
   DB93_DBX006_6 : BOOL ;
   DB93_DBX006_7 : BOOL ;
   DB93_DBX007_0 : BOOL ;
   DB93_DBX007_1 : BOOL ;
   DB93_DBX007_2 : BOOL ;
   DB93_DBX007_3 : BOOL ;
   DB93_DBX007_4 : BOOL ;
   DB93_DBX007_5 : BOOL ;
   DB93_DBX007_6 : BOOL ;
   DB93_DBX007_7 : BOOL ;
   DB93_DBX008_0 : BOOL ;
   DB93_DBX008_1 : BOOL ;
   DB93_DBX008_2 : BOOL ;
   DB93_DBX008_3 : BOOL ;
   DB93_DBX008_4 : BOOL ;
   DB93_DBX008_5 : BOOL ;
   DB93_DBX008_6 : BOOL ;
   DB93_DBX008_7 : BOOL ;
   DB93_DBX009_0 : BOOL ;
   DB93_DBX009_1 : BOOL ;
   DB93_DBX009_2 : BOOL ;
   DB93_DBX009_3 : BOOL ;
   DB93_DBX009_4 : BOOL ;
   DB93_DBX009_5 : BOOL ;
   DB93_DBX009_6 : BOOL ;
   DB93_DBX009_7 : BOOL ;
   DB93_DBX010_0 : BOOL ;
   DB93_DBX010_1 : BOOL ;
   DB93_DBX010_2 : BOOL ;
   DB93_DBX010_3 : BOOL ;
   DB93_DBX010_4 : BOOL ;
   DB93_DBX010_5 : BOOL ;
   DB93_DBX010_6 : BOOL ;
   DB93_DBX010_7 : BOOL ;
   DB93_DBX011_0 : BOOL ;
   DB93_DBX011_1 : BOOL ;
   DB93_DBX011_2 : BOOL ;
   DB93_DBX011_3 : BOOL ;
   DB93_DBX011_4 : BOOL ;
   DB93_DBX011_5 : BOOL ;
   DB93_DBX011_6 : BOOL ;
   DB93_DBX011_7 : BOOL ;
   DB93_DBX012_0 : BOOL ;
   DB93_DBX012_1 : BOOL ;
   DB93_DBX012_2 : BOOL ;
   DB93_DBX012_3 : BOOL ;
   DB93_DBX012_4 : BOOL ;
   DB93_DBX012_5 : BOOL ;
   DB93_DBX012_6 : BOOL ;
   DB93_DBX012_7 : BOOL ;
   DB93_DBX013_0 : BOOL ;
   DB93_DBX013_1 : BOOL ;
   DB93_DBX013_2 : BOOL ;
   DB93_DBX013_3 : BOOL ;
   DB93_DBX013_4 : BOOL ;
   DB93_DBX013_5 : BOOL ;
   DB93_DBX013_6 : BOOL ;
   DB93_DBX013_7 : BOOL ;
   DB93_DBX014_0 : BOOL ;
   DB93_DBX014_1 : BOOL ;
   DB93_DBX014_2 : BOOL ;
   DB93_DBX014_3 : BOOL ;
   DB93_DBX014_4 : BOOL ;
   DB93_DBX014_5 : BOOL ;
   DB93_DBX014_6 : BOOL ;
   DB93_DBX014_7 : BOOL ;
   DB93_DBX015_0 : BOOL ;
   DB93_DBX015_1 : BOOL ;
   DB93_DBX015_2 : BOOL ;
   DB93_DBX015_3 : BOOL ;
   DB93_DBX015_4 : BOOL ;
   DB93_DBX015_5 : BOOL ;
   DB93_DBX015_6 : BOOL ;
   DB93_DBX015_7 : BOOL ;
   DB93_DBX016_0 : BOOL ;
   DB93_DBX016_1 : BOOL ;
   DB93_DBX016_2 : BOOL ;
   DB93_DBX016_3 : BOOL ;
   DB93_DBX016_4 : BOOL ;
   DB93_DBX016_5 : BOOL ;
   DB93_DBX016_6 : BOOL ;
   DB93_DBX016_7 : BOOL ;
   DB93_DBX017_0 : BOOL ;
   DB93_DBX017_1 : BOOL ;
   DB93_DBX017_2 : BOOL ;
   DB93_DBX017_3 : BOOL ;
   DB93_DBX017_4 : BOOL ;
   DB93_DBX017_5 : BOOL ;
   DB93_DBX017_6 : BOOL ;
   DB93_DBX017_7 : BOOL ;
   DB93_DBX018_0 : BOOL ;	//Cage 24 preforming motor electric brake relay [-632K1|A004.0]
   DB93_DBX018_1 : BOOL ;	//Cage 24 preforming motor blower contactor [-632K2|A004.1]
   DB93_DBX018_2 : BOOL ;	//Cage 24 motor blower contactor [-632K3|A004.2]
   DB93_DBX018_3 : BOOL ;	//Cage 24 loading motor S rotation contactor [-632K4|A004.3]
   DB93_DBX018_4 : BOOL ;	//Cage 24 loading motor Z rotation contactor [-632K5|A004.4]
   DB93_DBX018_5 : BOOL ;
   DB93_DBX018_6 : BOOL ;	//Cage 24 guard  blower motor contactor [-632K7|A004.6]
   DB93_DBX018_7 : BOOL ;
   DB93_DBX019_0 : BOOL ;
   DB93_DBX019_1 : BOOL ;
   DB93_DBX019_2 : BOOL ;
   DB93_DBX019_3 : BOOL ;
   DB93_DBX019_4 : BOOL ;
   DB93_DBX019_5 : BOOL ;
   DB93_DBX019_6 : BOOL ;
   DB93_DBX019_7 : BOOL ;
   DB93_DBX020_0 : BOOL ;	//Cage 24 loading motor engaging electric valve [-682Y1|A042.0]
   DB93_DBX020_1 : BOOL ;	//Cage 24 loading motor disingaging electric valve [-682Y2|A042.1]
   DB93_DBX020_2 : BOOL ;	//Cage 24 cage block brake electric valve [-682Y3|A042.2]
   DB93_DBX020_3 : BOOL ;	//Cage 24 open air in cage electric valve [-683Y1|A042.3]
   DB93_DBX020_4 : BOOL ;	//Cage 24 close air in cage electric valve [-683Y2|A042.4]
   DB93_DBX020_5 : BOOL ;	//Cage 24 loading pinston engaging into cage electric valve [-683Y3|A042.5]
   DB93_DBX020_6 : BOOL ;	//Cage 24 loading pinston disengaging into cage electric valve [-683Y4|A042.6]
   DB93_DBX020_7 : BOOL ;	//Cage 24 pintles locking system opening electric valve [-684Y5|A042.7]
   DB93_DBX021_0 : BOOL ;	//Cage 24 pintles locking system closing electric valve [-684Y6|A043.0]
   DB93_DBX021_1 : BOOL ;	//Cage 24 pintles opening electric valve [-684Y7|A043.1]
   DB93_DBX021_2 : BOOL ;	//Cage 24 pintles closing electric valve [-684Y8|A043.2]
   DB93_DBX021_3 : BOOL ;	//Cage 24 front door locking [-686Y1:LOCK|A043.3]
   DB93_DBX021_4 : BOOL ;	//Cage 24 guard opening electric valve [-684Y3|A043.4]
   DB93_DBX021_5 : BOOL ;	//Cage 24 guard closing electric valve [-684Y4|A043.5]
   DB93_DBX021_6 : BOOL ;	//Cage 24 loading run pilot lamp [-663S3:LAMP|A043.6]
   DB93_DBX021_7 : BOOL ;	//Cage 24 loading insertion pilot lamp [-663S7:LAMP|A043.7]
   DB93_DBX022_0 : BOOL ;	//Cage 24 pintles open pilot lamp [-687H1:LAMP|A044.0]
   DB93_DBX022_1 : BOOL ;	//Cage 24 broken wire pilot lamp [-687H2:LAMP|A044.1]
   DB93_DBX022_2 : BOOL ;
   DB93_DBX022_3 : BOOL ;
   DB93_DBX022_4 : BOOL ;	//Cage 24 alarm reset pilot lamp [-663S4:LAMP|A044.4]
   DB93_DBX022_5 : BOOL ;
   DB93_DBX022_6 : BOOL ;
   DB93_DBX022_7 : BOOL ;
   DB93_DBX023_0 : BOOL ;
   DB93_DBX023_1 : BOOL ;
   DB93_DBX023_2 : BOOL ;
   DB93_DBX023_3 : BOOL ;
   DB93_DBX023_4 : BOOL ;	//Cage 24 preforming guard locking [-688Y8:LOCK|A045.4]
   DB93_DBX023_5 : BOOL ;
   DB93_DBX023_6 : BOOL ;
   DB93_DBX023_7 : BOOL ;
   DB93_DBX024_0 : BOOL ;	//Cage 24 stand by zone enable to loader [-MCB24:11|A007.4]
   DB93_DBX024_1 : BOOL ;	//Cage 24 presence of bobbins inside cage to loader [-MCB24:12|A007.5]
   DB93_DBX024_2 : BOOL ;	//Cage 24 loader lock piston inserted to loader [-MCB24:13|A007.6]
   DB93_DBX024_3 : BOOL ;	//Cage 24 open pintles to loader [-MCB24:14|A007.7]
   DB93_DBX024_4 : BOOL ;
   DB93_DBX024_5 : BOOL ;
   DB93_DBX024_6 : BOOL ;
   DB93_DBX024_7 : BOOL ;
   DB93_DBX025_0 : BOOL ;	//Cage 24 loader lock piston valve
   DB93_DBX025_1 : BOOL ;	//Cage 24 loader unlock piston valve
   DB93_DBX025_2 : BOOL ;
   DB93_DBX025_3 : BOOL ;
   DB93_DBX025_4 : BOOL ;
   DB93_DBX025_5 : BOOL ;
   DB93_DBX025_6 : BOOL ;
   DB93_DBX025_7 : BOOL ;
   DB93_DBX026_0 : BOOL ;
   DB93_DBX026_1 : BOOL ;
   DB93_DBX026_2 : BOOL ;
   DB93_DBX026_3 : BOOL ;
   DB93_DBX026_4 : BOOL ;
   DB93_DBX026_5 : BOOL ;
   DB93_DBX026_6 : BOOL ;
   DB93_DBX026_7 : BOOL ;
   DB93_DBX027_0 : BOOL ;
   DB93_DBX027_1 : BOOL ;
   DB93_DBX027_2 : BOOL ;
   DB93_DBX027_3 : BOOL ;
   DB93_DBX027_4 : BOOL ;
   DB93_DBX027_5 : BOOL ;
   DB93_DBX027_6 : BOOL ;
   DB93_DBX027_7 : BOOL ;
   DB93_DBX028_0 : BOOL ;	//Cage 18 preforming motor electric brake relay [-532K1|A000.7]
   DB93_DBX028_1 : BOOL ;	//Cage 18 preforming motor blower contactor [-532K2|A001.0]
   DB93_DBX028_2 : BOOL ;	//Cage 18 motor blower contactor [-532K3|A001.1]
   DB93_DBX028_3 : BOOL ;	//Cage 18 loading motor s rotation contactor [-532K4|A001.2]
   DB93_DBX028_4 : BOOL ;	//Cage 18 loading motor z rotation contactor [-532K5|A001.3]
   DB93_DBX028_5 : BOOL ;
   DB93_DBX028_6 : BOOL ;	//Cage 18 guard blower motor contactor [-532K7|A001.5]
   DB93_DBX028_7 : BOOL ;
   DB93_DBX029_0 : BOOL ;
   DB93_DBX029_1 : BOOL ;
   DB93_DBX029_2 : BOOL ;
   DB93_DBX029_3 : BOOL ;
   DB93_DBX029_4 : BOOL ;
   DB93_DBX029_5 : BOOL ;
   DB93_DBX029_6 : BOOL ;
   DB93_DBX029_7 : BOOL ;
   DB93_DBX030_0 : BOOL ;	//Cage 18 loading motor engaging electric valve [-582Y1|A052.0]
   DB93_DBX030_1 : BOOL ;	//Cage 18 loading motor disengaging electric valve [-582Y2|A052.1]
   DB93_DBX030_2 : BOOL ;	//Cage 18 block brake electric valve [-582Y3|A052.2]
   DB93_DBX030_3 : BOOL ;	//Cage 18 air inlet electric valve [-583Y1|A052.3]
   DB93_DBX030_4 : BOOL ;	//Cage 18 air outlet electric valve [-583Y2|A052.4]
   DB93_DBX030_5 : BOOL ;	//Cage 18 loading piston engaging into Cage electric valve [-583Y3|A052.5]
   DB93_DBX030_6 : BOOL ;	//Cage 18 loading piston disengaging from Cage electric valve [-583Y4|A052.6]
   DB93_DBX030_7 : BOOL ;	//Cage 18 pintles locking system opening electric valves [-584Y5|A052.7]
   DB93_DBX031_0 : BOOL ;	//Cage 18 pintles locking system closing electric valves [-584Y6|A053.0]
   DB93_DBX031_1 : BOOL ;	//Cage 18 pintles opening electric valves [-584Y7|A053.1]
   DB93_DBX031_2 : BOOL ;	//Cage 18 pintles closing electric valves [-584Y8|A053.2]
   DB93_DBX031_3 : BOOL ;	//Cage 18 front door locking [-586Y1:LOCK|A053.3]
   DB93_DBX031_4 : BOOL ;	//Cage 18 guard opening electric valve [-586Y3|A053.4]
   DB93_DBX031_5 : BOOL ;	//Cage 18 guard closing electric valve [-586Y4|A053.5]
   DB93_DBX031_6 : BOOL ;	//Cage 18 loading run pilot lamp [-563S3:LAMP|A053.6]
   DB93_DBX031_7 : BOOL ;	//Cage 18 loading insertion pilot lamp [-564S7:LAMP|A053.7]
   DB93_DBX032_0 : BOOL ;	//Cage 18 pintles open pilot lamp [-587H1|A054.0]
   DB93_DBX032_1 : BOOL ;	//Cage 18 broken wire pilot lamp [-587H2|A054.1]
   DB93_DBX032_2 : BOOL ;
   DB93_DBX032_3 : BOOL ;
   DB93_DBX032_4 : BOOL ;	//Cage 18 alarms reset pilot lamp [-563S4:LAMP|A054.4]
   DB93_DBX032_5 : BOOL ;
   DB93_DBX032_6 : BOOL ;
   DB93_DBX032_7 : BOOL ;
   DB93_DBX033_0 : BOOL ;
   DB93_DBX033_1 : BOOL ;
   DB93_DBX033_2 : BOOL ;
   DB93_DBX033_3 : BOOL ;
   DB93_DBX033_4 : BOOL ;	//Cage 18 preforming guard locking [-565Y8:LOCK|A055.4]
   DB93_DBX033_5 : BOOL ;
   DB93_DBX033_6 : BOOL ;
   DB93_DBX033_7 : BOOL ;
   DB93_DBX034_0 : BOOL ;	//Cage 18 stand by zone enable to loader [-MCB18:11|A007.0]
   DB93_DBX034_1 : BOOL ;	//Cage 18 presence of bobbins inside cage to loader [-MCB18:12|A007.1]
   DB93_DBX034_2 : BOOL ;	//Cage 18 loader lock piston inserted to loader [-MCB18:13|A007.2]
   DB93_DBX034_3 : BOOL ;	//Cage 18 open pintles to loader [-MCB18:14|A007.3]
   DB93_DBX034_4 : BOOL ;
   DB93_DBX034_5 : BOOL ;
   DB93_DBX034_6 : BOOL ;
   DB93_DBX034_7 : BOOL ;
   DB93_DBX035_0 : BOOL ;	//Cage 18 loader lock piston valve
   DB93_DBX035_1 : BOOL ;	//Cage 18 loader unlock piston valve
   DB93_DBX035_2 : BOOL ;
   DB93_DBX035_3 : BOOL ;
   DB93_DBX035_4 : BOOL ;
   DB93_DBX035_5 : BOOL ;
   DB93_DBX035_6 : BOOL ;
   DB93_DBX035_7 : BOOL ;
   DB93_DBX036_0 : BOOL ;
   DB93_DBX036_1 : BOOL ;
   DB93_DBX036_2 : BOOL ;
   DB93_DBX036_3 : BOOL ;
   DB93_DBX036_4 : BOOL ;
   DB93_DBX036_5 : BOOL ;
   DB93_DBX036_6 : BOOL ;
   DB93_DBX036_7 : BOOL ;
   DB93_DBX037_0 : BOOL ;
   DB93_DBX037_1 : BOOL ;
   DB93_DBX037_2 : BOOL ;
   DB93_DBX037_3 : BOOL ;
   DB93_DBX037_4 : BOOL ;
   DB93_DBX037_5 : BOOL ;
   DB93_DBX037_6 : BOOL ;
   DB93_DBX037_7 : BOOL ;
   DB93_DBX038_0 : BOOL ;	//Cage 12 preforming motor electric brake relay [-432K1|A001.6]
   DB93_DBX038_1 : BOOL ;	//Cage 12 preforming motor blower contactor [-432K2|A001.7]
   DB93_DBX038_2 : BOOL ;	//Cage 12 motor blower contactor [-432K3|A002.0]
   DB93_DBX038_3 : BOOL ;	//Cage 12 loading motor s rotation contactor [-432K4|A002.1]
   DB93_DBX038_4 : BOOL ;	//Cage 12 loading motor z rotation contactor [-432K5|A002.2]
   DB93_DBX038_5 : BOOL ;
   DB93_DBX038_6 : BOOL ;	//Cage 12 guard blower motor contactor [-432K7|A002.4]
   DB93_DBX038_7 : BOOL ;
   DB93_DBX039_0 : BOOL ;
   DB93_DBX039_1 : BOOL ;
   DB93_DBX039_2 : BOOL ;
   DB93_DBX039_3 : BOOL ;
   DB93_DBX039_4 : BOOL ;
   DB93_DBX039_5 : BOOL ;
   DB93_DBX039_6 : BOOL ;
   DB93_DBX039_7 : BOOL ;
   DB93_DBX040_0 : BOOL ;	//Cage 12 loading motor engaging electric valve [-482Y1|A062.0]
   DB93_DBX040_1 : BOOL ;	//Cage 12 loading motor disengaging electric valve [-482Y2|A062.1]
   DB93_DBX040_2 : BOOL ;	//Cage 12 block brake electric valve [-482Y3|A062.2]
   DB93_DBX040_3 : BOOL ;	//Cage 12 air inlet electric valve [-483Y1|A062.3]
   DB93_DBX040_4 : BOOL ;	//Cage 12 air outlet electric valve [-483Y2|A062.4]
   DB93_DBX040_5 : BOOL ;	//Cage 12 loading piston engaging into cage electric valve [-483Y3|A062.5]
   DB93_DBX040_6 : BOOL ;	//Cage 12 loading piston disengaging from cage electric valve [-483Y4|A062.6]
   DB93_DBX040_7 : BOOL ;	//Cage 12 pintles locking system opening electric valves [-484Y5|A062.7]
   DB93_DBX041_0 : BOOL ;	//Cage 12 pintles locking system closing electric valves [-484Y6|A063.0]
   DB93_DBX041_1 : BOOL ;	//Cage 12 pintles opening electric valves [-484Y7|A063.1]
   DB93_DBX041_2 : BOOL ;	//Cage 12 pintles closing electric valves [-484Y8|A063.2]
   DB93_DBX041_3 : BOOL ;	//Cage 12 front door locking [-486Y1:LOCK|A063.3]
   DB93_DBX041_4 : BOOL ;	//Cage 12 guard opening electric valve [-486Y3|A063.4]
   DB93_DBX041_5 : BOOL ;	//Cage 12 guard closing electric valve [-486Y4|A063.5]
   DB93_DBX041_6 : BOOL ;	//Cage 12 loading run pilot lamp [-463S3:LAMP|A063.6]
   DB93_DBX041_7 : BOOL ;	//Cage 12 loading insertion pilot lamp [-463S7:LAMP|A063.7]
   DB93_DBX042_0 : BOOL ;	//Cage 12 pintles open pilot lamp [-487H1:LAMP|A064.0]
   DB93_DBX042_1 : BOOL ;	//Cage 12 broken wire pilot lamp [-487H2:LAMP|A064.1]
   DB93_DBX042_2 : BOOL ;
   DB93_DBX042_3 : BOOL ;
   DB93_DBX042_4 : BOOL ;	//Cage 12 alarms reset pilot lamp [-463S4:LAMP|A064.4]
   DB93_DBX042_5 : BOOL ;
   DB93_DBX042_6 : BOOL ;
   DB93_DBX042_7 : BOOL ;
   DB93_DBX043_0 : BOOL ;
   DB93_DBX043_1 : BOOL ;
   DB93_DBX043_2 : BOOL ;
   DB93_DBX043_3 : BOOL ;
   DB93_DBX043_4 : BOOL ;	//Cage 12 preforming guard locking [-489Y8:LOCK|A065.4]
   DB93_DBX043_5 : BOOL ;
   DB93_DBX043_6 : BOOL ;
   DB93_DBX043_7 : BOOL ;
   DB93_DBX044_0 : BOOL ;	//Cage 12 stand by zone enable to loader [-MCB12:11|A006.4]
   DB93_DBX044_1 : BOOL ;	//Cage 12 presence of bobbins inside cage to loader [-MCB12:12|A006.5]
   DB93_DBX044_2 : BOOL ;	//Cage 12 loader lock piston inserted to loader [-MCB12:13|A006.6]
   DB93_DBX044_3 : BOOL ;	//Cage 12 open pintles to loader [-MCB12:14|A006.7]
   DB93_DBX044_4 : BOOL ;
   DB93_DBX044_5 : BOOL ;
   DB93_DBX044_6 : BOOL ;
   DB93_DBX044_7 : BOOL ;
   DB93_DBX045_0 : BOOL ;	//Cage 12 loader lock piston valve
   DB93_DBX045_1 : BOOL ;	//Cage 12 loader unlock piston valve
   DB93_DBX045_2 : BOOL ;
   DB93_DBX045_3 : BOOL ;
   DB93_DBX045_4 : BOOL ;
   DB93_DBX045_5 : BOOL ;
   DB93_DBX045_6 : BOOL ;
   DB93_DBX045_7 : BOOL ;
   DB93_DBX046_0 : BOOL ;
   DB93_DBX046_1 : BOOL ;
   DB93_DBX046_2 : BOOL ;
   DB93_DBX046_3 : BOOL ;
   DB93_DBX046_4 : BOOL ;
   DB93_DBX046_5 : BOOL ;
   DB93_DBX046_6 : BOOL ;
   DB93_DBX046_7 : BOOL ;
   DB93_DBX047_0 : BOOL ;
   DB93_DBX047_1 : BOOL ;
   DB93_DBX047_2 : BOOL ;
   DB93_DBX047_3 : BOOL ;
   DB93_DBX047_4 : BOOL ;
   DB93_DBX047_5 : BOOL ;
   DB93_DBX047_6 : BOOL ;
   DB93_DBX047_7 : BOOL ;
   DB93_DBX048_0 : BOOL ;
   DB93_DBX048_1 : BOOL ;
   DB93_DBX048_2 : BOOL ;	//Cage 6 motor blower contactor [-332K1|A002.5]
   DB93_DBX048_3 : BOOL ;	//Cage 6 loading motor s rotation contactor [-332K2|A002.6]
   DB93_DBX048_4 : BOOL ;	//Cage 6 loading motor z rotation contactor [-332K3|A002.7]
   DB93_DBX048_5 : BOOL ;
   DB93_DBX048_6 : BOOL ;	//Cage 6 guard blower motor contactor [-332K5|A003.1]
   DB93_DBX048_7 : BOOL ;
   DB93_DBX049_0 : BOOL ;
   DB93_DBX049_1 : BOOL ;
   DB93_DBX049_2 : BOOL ;
   DB93_DBX049_3 : BOOL ;
   DB93_DBX049_4 : BOOL ;
   DB93_DBX049_5 : BOOL ;
   DB93_DBX049_6 : BOOL ;
   DB93_DBX049_7 : BOOL ;
   DB93_DBX050_0 : BOOL ;	//Cage 6 loading motor engaging electric valve [-382Y1|A072.0]
   DB93_DBX050_1 : BOOL ;	//Cage 6 loading motor disengaging electric valve [-382Y2|A072.1]
   DB93_DBX050_2 : BOOL ;	//Cage 6 block stationary brake electric valve [-382Y3|A072.2]
   DB93_DBX050_3 : BOOL ;	//Cage 6 air inlet electric valve [-383Y1|A072.3]
   DB93_DBX050_4 : BOOL ;	//Cage 6 air outlet electric valve [-383Y2|A072.4]
   DB93_DBX050_5 : BOOL ;	//Cage 6 loading piston engaging into cage electric valve [-383Y3|A072.5]
   DB93_DBX050_6 : BOOL ;	//Cage 6 loading piston disengaging from cage electric valve [-383Y4|A072.6]
   DB93_DBX050_7 : BOOL ;	//Cage 6 pintles locking system opening electric valves [-384K1|A072.7]
   DB93_DBX051_0 : BOOL ;	//Cage 6 pintles locking system closing electric valves [-384K2|A073.0]
   DB93_DBX051_1 : BOOL ;	//Cage 6 pintles opening electric valves [-384K3|A073.1]
   DB93_DBX051_2 : BOOL ;	//Cage 6 pintles closing electric valves [-384K4|A073.2]
   DB93_DBX051_3 : BOOL ;	//Cage 6 front door locking [-386Y1:LOCK|A073.3]
   DB93_DBX051_4 : BOOL ;	//Cage 6 guard opening electric valve [-386Y3|A073.4]
   DB93_DBX051_5 : BOOL ;	//Cage 6 guard closing electric valve [-386Y4|A073.5]
   DB93_DBX051_6 : BOOL ;	//Cage 6 loading run pilot lamp [-363S3:LAMP|A073.6]
   DB93_DBX051_7 : BOOL ;	//Cage 6 loading insertion pilot lamp [-364S7:LAMP|A073.7]
   DB93_DBX052_0 : BOOL ;	//Cage 6 pintles open pilot lamp [-387H1:LAMP|A074.0]
   DB93_DBX052_1 : BOOL ;	//Cage 6 broken wire pilot lamp [-387H2:LAMP|A074.1]
   DB93_DBX052_2 : BOOL ;
   DB93_DBX052_3 : BOOL ;
   DB93_DBX052_4 : BOOL ;	//Cage 6 alarms reset pilot lamp [-363S4:LAMP|A074.4]
   DB93_DBX052_5 : BOOL ;
   DB93_DBX052_6 : BOOL ;
   DB93_DBX052_7 : BOOL ;
   DB93_DBX053_0 : BOOL ;
   DB93_DBX053_1 : BOOL ;
   DB93_DBX053_2 : BOOL ;
   DB93_DBX053_3 : BOOL ;
   DB93_DBX053_4 : BOOL ;	//Cage 6 preforming guard locking [-388Y8|A075.4]
   DB93_DBX053_5 : BOOL ;
   DB93_DBX053_6 : BOOL ;
   DB93_DBX053_7 : BOOL ;
   DB93_DBX054_0 : BOOL ;	//Cage 6 stand by zone enable to loader [-MCB06:11|A006.0]
   DB93_DBX054_1 : BOOL ;	//Cage 6 presence of bobbins inside cage to loader [-MCB06:12|A006.1]
   DB93_DBX054_2 : BOOL ;	//Cage 6 loader lock piston inserted to loader [-MCB06:13|A006.2]
   DB93_DBX054_3 : BOOL ;	//Cage 6 open pintles to loader [-MCB06:14|A006.3]
   DB93_DBX054_4 : BOOL ;
   DB93_DBX054_5 : BOOL ;
   DB93_DBX054_6 : BOOL ;
   DB93_DBX054_7 : BOOL ;
   DB93_DBX055_0 : BOOL ;	//Cage 6 loader lock piston valve
   DB93_DBX055_1 : BOOL ;	//Cage 6 loader unlock piston valve
   DB93_DBX055_2 : BOOL ;
   DB93_DBX055_3 : BOOL ;
   DB93_DBX055_4 : BOOL ;
   DB93_DBX055_5 : BOOL ;
   DB93_DBX055_6 : BOOL ;
   DB93_DBX055_7 : BOOL ;
   DB93_DBX056_0 : BOOL ;
   DB93_DBX056_1 : BOOL ;
   DB93_DBX056_2 : BOOL ;
   DB93_DBX056_3 : BOOL ;
   DB93_DBX056_4 : BOOL ;
   DB93_DBX056_5 : BOOL ;
   DB93_DBX056_6 : BOOL ;
   DB93_DBX056_7 : BOOL ;
   DB93_DBX057_0 : BOOL ;
   DB93_DBX057_1 : BOOL ;
   DB93_DBX057_2 : BOOL ;
   DB93_DBX057_3 : BOOL ;
   DB93_DBX057_4 : BOOL ;
   DB93_DBX057_5 : BOOL ;
   DB93_DBX057_6 : BOOL ;
   DB93_DBX057_7 : BOOL ;
   DB93_DBX058_0 : BOOL ;	//Central Pay-off 630 broken wire pilot lamp [-390H1:LAMP|A075.5]
   DB93_DBX058_1 : BOOL ;	//Central Pay-off 630 pintle open pilot lamp [-390H2:LAMP|A075.6]
   DB93_DBX058_2 : BOOL ;	//Central Pay-off 630 pintle enable [-390K3|A075.7]
   DB93_DBX058_3 : BOOL ;
   DB93_DBX058_4 : BOOL ;
   DB93_DBX058_5 : BOOL ;
   DB93_DBX058_6 : BOOL ;
   DB93_DBX058_7 : BOOL ;
   DB93_DBX059_0 : BOOL ;
   DB93_DBX059_1 : BOOL ;
   DB93_DBX059_2 : BOOL ;
   DB93_DBX059_3 : BOOL ;
   DB93_DBX059_4 : BOOL ;
   DB93_DBX059_5 : BOOL ;
   DB93_DBX059_6 : BOOL ;
   DB93_DBX059_7 : BOOL ;
   DB93_DBX060_0 : BOOL ;
   DB93_DBX060_1 : BOOL ;
   DB93_DBX060_2 : BOOL ;
   DB93_DBX060_3 : BOOL ;
   DB93_DBX060_4 : BOOL ;
   DB93_DBX060_5 : BOOL ;
   DB93_DBX060_6 : BOOL ;
   DB93_DBX060_7 : BOOL ;
   DB93_DBX061_0 : BOOL ;
   DB93_DBX061_1 : BOOL ;
   DB93_DBX061_2 : BOOL ;
   DB93_DBX061_3 : BOOL ;
   DB93_DBX061_4 : BOOL ;
   DB93_DBX061_5 : BOOL ;
   DB93_DBX061_6 : BOOL ;
   DB93_DBX061_7 : BOOL ;
   DB93_DBX062_0 : BOOL ;
   DB93_DBX062_1 : BOOL ;
   DB93_DBX062_2 : BOOL ;
   DB93_DBX062_3 : BOOL ;
   DB93_DBX062_4 : BOOL ;
   DB93_DBX062_5 : BOOL ;
   DB93_DBX062_6 : BOOL ;
   DB93_DBX062_7 : BOOL ;
   DB93_DBX063_0 : BOOL ;
   DB93_DBX063_1 : BOOL ;
   DB93_DBX063_2 : BOOL ;
   DB93_DBX063_3 : BOOL ;
   DB93_DBX063_4 : BOOL ;
   DB93_DBX063_5 : BOOL ;
   DB93_DBX063_6 : BOOL ;
   DB93_DBX063_7 : BOOL ;
   DB93_DBX064_0 : BOOL ;
   DB93_DBX064_1 : BOOL ;
   DB93_DBX064_2 : BOOL ;
   DB93_DBX064_3 : BOOL ;
   DB93_DBX064_4 : BOOL ;
   DB93_DBX064_5 : BOOL ;
   DB93_DBX064_6 : BOOL ;
   DB93_DBX064_7 : BOOL ;
   DB93_DBX065_0 : BOOL ;
   DB93_DBX065_1 : BOOL ;
   DB93_DBX065_2 : BOOL ;
   DB93_DBX065_3 : BOOL ;
   DB93_DBX065_4 : BOOL ;
   DB93_DBX065_5 : BOOL ;
   DB93_DBX065_6 : BOOL ;
   DB93_DBX065_7 : BOOL ;
   DB93_DBX066_0 : BOOL ;
   DB93_DBX066_1 : BOOL ;
   DB93_DBX066_2 : BOOL ;
   DB93_DBX066_3 : BOOL ;
   DB93_DBX066_4 : BOOL ;
   DB93_DBX066_5 : BOOL ;
   DB93_DBX066_6 : BOOL ;
   DB93_DBX066_7 : BOOL ;
   DB93_DBX067_0 : BOOL ;
   DB93_DBX067_1 : BOOL ;
   DB93_DBX067_2 : BOOL ;
   DB93_DBX067_3 : BOOL ;
   DB93_DBX067_4 : BOOL ;
   DB93_DBX067_5 : BOOL ;
   DB93_DBX067_6 : BOOL ;
   DB93_DBX067_7 : BOOL ;
   DB93_DBX068_0 : BOOL ;
   DB93_DBX068_1 : BOOL ;
   DB93_DBX068_2 : BOOL ;
   DB93_DBX068_3 : BOOL ;
   DB93_DBX068_4 : BOOL ;
   DB93_DBX068_5 : BOOL ;
   DB93_DBX068_6 : BOOL ;
   DB93_DBX068_7 : BOOL ;
   DB93_DBX069_0 : BOOL ;
   DB93_DBX069_1 : BOOL ;
   DB93_DBX069_2 : BOOL ;
   DB93_DBX069_3 : BOOL ;
   DB93_DBX069_4 : BOOL ;
   DB93_DBX069_5 : BOOL ;
   DB93_DBX069_6 : BOOL ;
   DB93_DBX069_7 : BOOL ;
   DB93_DBX070_0 : BOOL ;
   DB93_DBX070_1 : BOOL ;
   DB93_DBX070_2 : BOOL ;
   DB93_DBX070_3 : BOOL ;
   DB93_DBX070_4 : BOOL ;
   DB93_DBX070_5 : BOOL ;
   DB93_DBX070_6 : BOOL ;
   DB93_DBX070_7 : BOOL ;
   DB93_DBX071_0 : BOOL ;
   DB93_DBX071_1 : BOOL ;
   DB93_DBX071_2 : BOOL ;
   DB93_DBX071_3 : BOOL ;
   DB93_DBX071_4 : BOOL ;
   DB93_DBX071_5 : BOOL ;
   DB93_DBX071_6 : BOOL ;
   DB93_DBX071_7 : BOOL ;
   DB93_DBX072_0 : BOOL ;
   DB93_DBX072_1 : BOOL ;
   DB93_DBX072_2 : BOOL ;
   DB93_DBX072_3 : BOOL ;
   DB93_DBX072_4 : BOOL ;
   DB93_DBX072_5 : BOOL ;
   DB93_DBX072_6 : BOOL ;
   DB93_DBX072_7 : BOOL ;
   DB93_DBX073_0 : BOOL ;
   DB93_DBX073_1 : BOOL ;
   DB93_DBX073_2 : BOOL ;
   DB93_DBX073_3 : BOOL ;
   DB93_DBX073_4 : BOOL ;
   DB93_DBX073_5 : BOOL ;
   DB93_DBX073_6 : BOOL ;
   DB93_DBX073_7 : BOOL ;
   DB93_DBX074_0 : BOOL ;
   DB93_DBX074_1 : BOOL ;
   DB93_DBX074_2 : BOOL ;
   DB93_DBX074_3 : BOOL ;
   DB93_DBX074_4 : BOOL ;
   DB93_DBX074_5 : BOOL ;
   DB93_DBX074_6 : BOOL ;
   DB93_DBX074_7 : BOOL ;
   DB93_DBX075_0 : BOOL ;
   DB93_DBX075_1 : BOOL ;
   DB93_DBX075_2 : BOOL ;
   DB93_DBX075_3 : BOOL ;
   DB93_DBX075_4 : BOOL ;
   DB93_DBX075_5 : BOOL ;
   DB93_DBX075_6 : BOOL ;
   DB93_DBX075_7 : BOOL ;
   DB93_DBX076_0 : BOOL ;
   DB93_DBX076_1 : BOOL ;
   DB93_DBX076_2 : BOOL ;
   DB93_DBX076_3 : BOOL ;
   DB93_DBX076_4 : BOOL ;
   DB93_DBX076_5 : BOOL ;
   DB93_DBX076_6 : BOOL ;
   DB93_DBX076_7 : BOOL ;
   DB93_DBX077_0 : BOOL ;
   DB93_DBX077_1 : BOOL ;
   DB93_DBX077_2 : BOOL ;
   DB93_DBX077_3 : BOOL ;
   DB93_DBX077_4 : BOOL ;
   DB93_DBX077_5 : BOOL ;
   DB93_DBX077_6 : BOOL ;
   DB93_DBX077_7 : BOOL ;
   DB93_DBX078_0 : BOOL ;
   DB93_DBX078_1 : BOOL ;
   DB93_DBX078_2 : BOOL ;
   DB93_DBX078_3 : BOOL ;
   DB93_DBX078_4 : BOOL ;
   DB93_DBX078_5 : BOOL ;
   DB93_DBX078_6 : BOOL ;
   DB93_DBX078_7 : BOOL ;
   DB93_DBX079_0 : BOOL ;
   DB93_DBX079_1 : BOOL ;
   DB93_DBX079_2 : BOOL ;
   DB93_DBX079_3 : BOOL ;
   DB93_DBX079_4 : BOOL ;
   DB93_DBX079_5 : BOOL ;
   DB93_DBX079_6 : BOOL ;
   DB93_DBX079_7 : BOOL ;
   DB93_DBX080_0 : BOOL ;
   DB93_DBX080_1 : BOOL ;
   DB93_DBX080_2 : BOOL ;
   DB93_DBX080_3 : BOOL ;
   DB93_DBX080_4 : BOOL ;
   DB93_DBX080_5 : BOOL ;
   DB93_DBX080_6 : BOOL ;
   DB93_DBX080_7 : BOOL ;
   DB93_DBX081_0 : BOOL ;
   DB93_DBX081_1 : BOOL ;
   DB93_DBX081_2 : BOOL ;
   DB93_DBX081_3 : BOOL ;
   DB93_DBX081_4 : BOOL ;
   DB93_DBX081_5 : BOOL ;
   DB93_DBX081_6 : BOOL ;
   DB93_DBX081_7 : BOOL ;
   DB93_DBX082_0 : BOOL ;
   DB93_DBX082_1 : BOOL ;
   DB93_DBX082_2 : BOOL ;
   DB93_DBX082_3 : BOOL ;
   DB93_DBX082_4 : BOOL ;
   DB93_DBX082_5 : BOOL ;
   DB93_DBX082_6 : BOOL ;
   DB93_DBX082_7 : BOOL ;
   DB93_DBX083_0 : BOOL ;
   DB93_DBX083_1 : BOOL ;
   DB93_DBX083_2 : BOOL ;
   DB93_DBX083_3 : BOOL ;
   DB93_DBX083_4 : BOOL ;
   DB93_DBX083_5 : BOOL ;
   DB93_DBX083_6 : BOOL ;
   DB93_DBX083_7 : BOOL ;
   DB93_DBX084_0 : BOOL ;
   DB93_DBX084_1 : BOOL ;
   DB93_DBX084_2 : BOOL ;
   DB93_DBX084_3 : BOOL ;
   DB93_DBX084_4 : BOOL ;
   DB93_DBX084_5 : BOOL ;
   DB93_DBX084_6 : BOOL ;
   DB93_DBX084_7 : BOOL ;
   DB93_DBX085_0 : BOOL ;
   DB93_DBX085_1 : BOOL ;
   DB93_DBX085_2 : BOOL ;
   DB93_DBX085_3 : BOOL ;
   DB93_DBX085_4 : BOOL ;
   DB93_DBX085_5 : BOOL ;
   DB93_DBX085_6 : BOOL ;
   DB93_DBX085_7 : BOOL ;
   DB93_DBX086_0 : BOOL ;
   DB93_DBX086_1 : BOOL ;
   DB93_DBX086_2 : BOOL ;
   DB93_DBX086_3 : BOOL ;
   DB93_DBX086_4 : BOOL ;
   DB93_DBX086_5 : BOOL ;
   DB93_DBX086_6 : BOOL ;
   DB93_DBX086_7 : BOOL ;
   DB93_DBX087_0 : BOOL ;
   DB93_DBX087_1 : BOOL ;
   DB93_DBX087_2 : BOOL ;
   DB93_DBX087_3 : BOOL ;
   DB93_DBX087_4 : BOOL ;
   DB93_DBX087_5 : BOOL ;
   DB93_DBX087_6 : BOOL ;
   DB93_DBX087_7 : BOOL ;
   DB93_DBX088_0 : BOOL ;
   DB93_DBX088_1 : BOOL ;
   DB93_DBX088_2 : BOOL ;
   DB93_DBX088_3 : BOOL ;
   DB93_DBX088_4 : BOOL ;
   DB93_DBX088_5 : BOOL ;
   DB93_DBX088_6 : BOOL ;
   DB93_DBX088_7 : BOOL ;
   DB93_DBX089_0 : BOOL ;
   DB93_DBX089_1 : BOOL ;
   DB93_DBX089_2 : BOOL ;
   DB93_DBX089_3 : BOOL ;
   DB93_DBX089_4 : BOOL ;
   DB93_DBX089_5 : BOOL ;
   DB93_DBX089_6 : BOOL ;
   DB93_DBX089_7 : BOOL ;
   DB93_DBX090_0 : BOOL ;
   DB93_DBX090_1 : BOOL ;
   DB93_DBX090_2 : BOOL ;
   DB93_DBX090_3 : BOOL ;
   DB93_DBX090_4 : BOOL ;
   DB93_DBX090_5 : BOOL ;
   DB93_DBX090_6 : BOOL ;
   DB93_DBX090_7 : BOOL ;
   DB93_DBX091_0 : BOOL ;
   DB93_DBX091_1 : BOOL ;
   DB93_DBX091_2 : BOOL ;
   DB93_DBX091_3 : BOOL ;
   DB93_DBX091_4 : BOOL ;
   DB93_DBX091_5 : BOOL ;
   DB93_DBX091_6 : BOOL ;
   DB93_DBX091_7 : BOOL ;
   DB93_DBX092_0 : BOOL ;
   DB93_DBX092_1 : BOOL ;
   DB93_DBX092_2 : BOOL ;
   DB93_DBX092_3 : BOOL ;
   DB93_DBX092_4 : BOOL ;
   DB93_DBX092_5 : BOOL ;
   DB93_DBX092_6 : BOOL ;
   DB93_DBX092_7 : BOOL ;
   DB93_DBX093_0 : BOOL ;
   DB93_DBX093_1 : BOOL ;
   DB93_DBX093_2 : BOOL ;
   DB93_DBX093_3 : BOOL ;
   DB93_DBX093_4 : BOOL ;
   DB93_DBX093_5 : BOOL ;
   DB93_DBX093_6 : BOOL ;
   DB93_DBX093_7 : BOOL ;
   DB93_DBX094_0 : BOOL ;
   DB93_DBX094_1 : BOOL ;
   DB93_DBX094_2 : BOOL ;
   DB93_DBX094_3 : BOOL ;
   DB93_DBX094_4 : BOOL ;
   DB93_DBX094_5 : BOOL ;
   DB93_DBX094_6 : BOOL ;
   DB93_DBX094_7 : BOOL ;
   DB93_DBX095_0 : BOOL ;
   DB93_DBX095_1 : BOOL ;
   DB93_DBX095_2 : BOOL ;
   DB93_DBX095_3 : BOOL ;
   DB93_DBX095_4 : BOOL ;
   DB93_DBX095_5 : BOOL ;
   DB93_DBX095_6 : BOOL ;
   DB93_DBX095_7 : BOOL ;
   DB93_DBX096_0 : BOOL ;
   DB93_DBX096_1 : BOOL ;
   DB93_DBX096_2 : BOOL ;
   DB93_DBX096_3 : BOOL ;
   DB93_DBX096_4 : BOOL ;
   DB93_DBX096_5 : BOOL ;
   DB93_DBX096_6 : BOOL ;
   DB93_DBX096_7 : BOOL ;
   DB93_DBX097_0 : BOOL ;
   DB93_DBX097_1 : BOOL ;
   DB93_DBX097_2 : BOOL ;
   DB93_DBX097_3 : BOOL ;
   DB93_DBX097_4 : BOOL ;
   DB93_DBX097_5 : BOOL ;
   DB93_DBX097_6 : BOOL ;
   DB93_DBX097_7 : BOOL ;
   DB93_DBX098_0 : BOOL ;
   DB93_DBX098_1 : BOOL ;
   DB93_DBX098_2 : BOOL ;
   DB93_DBX098_3 : BOOL ;
   DB93_DBX098_4 : BOOL ;
   DB93_DBX098_5 : BOOL ;
   DB93_DBX098_6 : BOOL ;
   DB93_DBX098_7 : BOOL ;
   DB93_DBX099_0 : BOOL ;
   DB93_DBX099_1 : BOOL ;
   DB93_DBX099_2 : BOOL ;
   DB93_DBX099_3 : BOOL ;
   DB93_DBX099_4 : BOOL ;
   DB93_DBX099_5 : BOOL ;
   DB93_DBX099_6 : BOOL ;
   DB93_DBX099_7 : BOOL ;
  END_STRUCT ;	
BEGIN
   DB93_DBX000_6 := TRUE;
   DB93_DBX001_3 := TRUE;
   DB93_DBX002_0 := TRUE;
   DB93_DBX004_6 := TRUE;
   DB93_DBX005_1 := TRUE;
   DB93_DBX005_2 := TRUE;
   DB93_DBX006_0 := TRUE;
   DB93_DBX006_2 := TRUE;
   DB93_DBX021_3 := TRUE;
   DB93_DBX021_7 := TRUE;
   DB93_DBX024_0 := TRUE;
   DB93_DBX024_2 := TRUE;
   DB93_DBX025_1 := TRUE;
   DB93_DBX031_3 := TRUE;
   DB93_DBX031_7 := TRUE;
   DB93_DBX034_0 := TRUE;
   DB93_DBX034_2 := TRUE;
   DB93_DBX035_1 := TRUE;
   DB93_DBX041_3 := TRUE;
   DB93_DBX044_2 := TRUE;
   DB93_DBX051_3 := TRUE;
   DB93_DBX058_2 := TRUE;
END_DATA_BLOCK

